   1:L PR[91] R[100]mm/sec CNT100;
   1:  PR[91,1] = PR[90,1] + 14.999;
   1:  PR[91,2] = PR[90,2] + -17.713;
   1:  PR[91,3] = PR[90,3] + 29.369;
   1:L PR[91] R[100]mm/sec CNT100;
   1:  PR[91,1] = PR[90,1] + 15.996;
   1:  PR[91,2] = PR[90,2] + -17.584;
   1:  PR[91,3] = PR[90,3] + 29.377;
   1:L PR[91] R[100]mm/sec CNT100;
   1:  PR[91,1] = PR[90,1] + 16.467;
   1:  PR[91,2] = PR[90,2] + -17.502;
   1:  PR[91,3] = PR[90,3] + 29.385;
   1:L PR[91] R[100]mm/sec CNT100;
   1:  PR[91,1] = PR[90,1] + 16.980;
   1:  PR[91,2] = PR[90,2] + -17.408;
   1:  PR[91,3] = PR[90,3] + 29.388;
   1:L PR[91] R[100]mm/sec CNT100;
   1:  PR[91,1] = PR[90,1] + 17.954;
   1:  PR[91,2] = PR[90,2] + -17.183;
   1:  PR[91,3] = PR[90,3] + 29.392;
   1:L PR[91] R[100]mm/sec CNT100;
   1:  PR[91,1] = PR[90,1] + 18.912;
   1:  PR[91,2] = PR[90,2] + -16.912;
   1:  PR[91,3] = PR[90,3] + 29.400;
   1:L PR[91] R[100]mm/sec CNT100;
   1:  PR[91,1] = PR[90,1] + 19.853;
   1:  PR[91,2] = PR[90,2] + -16.596;
   1:  PR[91,3] = PR[90,3] + 29.408;
   1:L PR[91] R[100]mm/sec CNT100;
   1:  PR[91,1] = PR[90,1] + 20.773;
   1:  PR[91,2] = PR[90,2] + -16.236;
   1:  PR[91,3] = PR[90,3] + 29.415;
   1:L PR[91] R[100]mm/sec CNT100;
   1:  PR[91,1] = PR[90,1] + 21.671;
   1:  PR[91,2] = PR[90,2] + -15.834;
   1:  PR[91,3] = PR[90,3] + 29.423;
   1:L PR[91] R[100]mm/sec CNT100;
   1:  PR[91,1] = PR[90,1] + 22.552;
   1:  PR[91,2] = PR[90,2] + -15.387;
   1:  PR[91,3] = PR[90,3] + 29.430;
   1:L PR[91] R[100]mm/sec CNT100;
   1:  PR[91,1] = PR[90,1] + 23.431;
   1:  PR[91,2] = PR[90,2] + -14.885;
   1:  PR[91,3] = PR[90,3] + 29.438;
   1:L PR[91] R[100]mm/sec CNT100;
   1:  PR[91,1] = PR[90,1] + 24.148;
   1:  PR[91,2] = PR[90,2] + -14.431;
   1:  PR[91,3] = PR[90,3] + 29.446;
   1:L PR[91] R[100]mm/sec CNT100;
   1:  PR[91,1] = PR[90,1] + 24.918;
   1:  PR[91,2] = PR[90,2] + -13.893;
   1:  PR[91,3] = PR[90,3] + 29.452;
   1:L PR[91] R[100]mm/sec CNT100;
   1:  PR[91,1] = PR[90,1] + 25.658;
   1:  PR[91,2] = PR[90,2] + -13.318;
   1:  PR[91,3] = PR[90,3] + 29.459;
   1:L PR[91] R[100]mm/sec CNT100;
   1:  PR[91,1] = PR[90,1] + 26.370;
   1:  PR[91,2] = PR[90,2] + -12.708;
   1:  PR[91,3] = PR[90,3] + 29.466;
   1:L PR[91] R[100]mm/sec CNT100;
   1:  PR[91,1] = PR[90,1] + 27.049;
   1:  PR[91,2] = PR[90,2] + -12.063;
   1:  PR[91,3] = PR[90,3] + 29.474;
   1:L PR[91] R[100]mm/sec CNT100;
   1:  PR[91,1] = PR[90,1] + 27.695;
   1:  PR[91,2] = PR[90,2] + -11.384;
   1:  PR[91,3] = PR[90,3] + 29.481;
   1:L PR[91] R[100]mm/sec CNT100;
   1:  PR[91,1] = PR[90,1] + 28.305;
   1:  PR[91,2] = PR[90,2] + -10.672;
   1:  PR[91,3] = PR[90,3] + 29.488;
   1:L PR[91] R[100]mm/sec CNT100;
   1:  PR[91,1] = PR[90,1] + 28.879;
   1:  PR[91,2] = PR[90,2] + -9.929;
   1:  PR[91,3] = PR[90,3] + 29.495;
   1:L PR[91] R[100]mm/sec CNT100;
   1:  PR[91,1] = PR[90,1] + 29.413;
   1:  PR[91,2] = PR[90,2] + -9.158;
   1:  PR[91,3] = PR[90,3] + 29.502;
   1:L PR[91] R[100]mm/sec CNT100;
   1:  PR[91,1] = PR[90,1] + 29.908;
   1:  PR[91,2] = PR[90,2] + -8.363;
   1:  PR[91,3] = PR[90,3] + 29.509;
   1:L PR[91] R[100]mm/sec CNT100;
   1:  PR[91,1] = PR[90,1] + 30.361;
   1:  PR[91,2] = PR[90,2] + -7.547;
   1:  PR[91,3] = PR[90,3] + 29.517;
   1:L PR[91] R[100]mm/sec CNT100;
   1:  PR[91,1] = PR[90,1] + 30.770;
   1:  PR[91,2] = PR[90,2] + -6.718;
   1:  PR[91,3] = PR[90,3] + 29.524;
   1:L PR[91] R[100]mm/sec CNT100;
   1:  PR[91,1] = PR[90,1] + 31.135;
   1:  PR[91,2] = PR[90,2] + -5.878;
   1:  PR[91,3] = PR[90,3] + 29.531;
   1:L PR[91] R[100]mm/sec CNT100;
   1:  PR[91,1] = PR[90,1] + 31.452;
   1:  PR[91,2] = PR[90,2] + -5.031;
   1:  PR[91,3] = PR[90,3] + 29.538;
   1:L PR[91] R[100]mm/sec CNT100;
   1:  PR[91,1] = PR[90,1] + 31.722;
   1:  PR[91,2] = PR[90,2] + -4.174;
   1:  PR[91,3] = PR[90,3] + 29.545;
   1:L PR[91] R[100]mm/sec CNT100;
   1:  PR[91,1] = PR[90,1] + 31.943;
   1:  PR[91,2] = PR[90,2] + -3.305;
   1:  PR[91,3] = PR[90,3] + 29.552;
   1:L PR[91] R[100]mm/sec CNT100;
   1:  PR[91,1] = PR[90,1] + 32.116;
   1:  PR[91,2] = PR[90,2] + -2.416;
   1:  PR[91,3] = PR[90,3] + 29.559;
   1:L PR[91] R[100]mm/sec CNT100;
   1:  PR[91,1] = PR[90,1] + 32.241;
   1:  PR[91,2] = PR[90,2] + -1.502;
   1:  PR[91,3] = PR[90,3] + 29.566;
   1:L PR[91] R[100]mm/sec CNT100;
   1:  PR[91,1] = PR[90,1] + 32.316;
   1:  PR[91,2] = PR[90,2] + -0.556;
   1:  PR[91,3] = PR[90,3] + 29.573;
   1:L PR[91] R[100]mm/sec CNT100;
   1:  PR[91,1] = PR[90,1] + 32.341;
   1:  PR[91,2] = PR[90,2] + 0.428;
   1:  PR[91,3] = PR[90,3] + 29.580;
   1:L PR[91] R[100]mm/sec CNT100;
   1:  PR[91,1] = PR[90,1] + 32.316;
   1:  PR[91,2] = PR[90,2] + 1.411;
   1:  PR[91,3] = PR[90,3] + 29.587;
   1:L PR[91] R[100]mm/sec CNT100;
   1:  PR[91,1] = PR[90,1] + 32.241;
   1:  PR[91,2] = PR[90,2] + 2.357;
   1:  PR[91,3] = PR[90,3] + 29.595;
   1:L PR[91] R[100]mm/sec CNT100;
   1:  PR[91,1] = PR[90,1] + 32.116;
   1:  PR[91,2] = PR[90,2] + 3.272;
   1:  PR[91,3] = PR[90,3] + 29.602;
   1:L PR[91] R[100]mm/sec CNT100;
   1:  PR[91,1] = PR[90,1] + 31.943;
   1:  PR[91,2] = PR[90,2] + 4.160;
   1:  PR[91,3] = PR[90,3] + 29.609;
   1:L PR[91] R[100]mm/sec CNT100;
   1:  PR[91,1] = PR[90,1] + 31.721;
   1:  PR[91,2] = PR[90,2] + 5.030;
   1:  PR[91,3] = PR[90,3] + 29.616;
   1:L PR[91] R[100]mm/sec CNT100;
   1:  PR[91,1] = PR[90,1] + 31.452;
   1:  PR[91,2] = PR[90,2] + 5.886;
   1:  PR[91,3] = PR[90,3] + 29.623;
   1:L PR[91] R[100]mm/sec CNT100;
   1:  PR[91,1] = PR[90,1] + 31.135;
   1:  PR[91,2] = PR[90,2] + 6.731;
   1:  PR[91,3] = PR[90,3] + 29.630;
   1:L PR[91] R[100]mm/sec CNT100;
   1:  PR[91,1] = PR[90,1] + 30.663;
   1:  PR[91,2] = PR[90,2] + 7.794;
   1:  PR[91,3] = PR[90,3] + 29.637;
   1:L PR[91] R[100]mm/sec CNT100;
   1:  PR[91,1] = PR[90,1] + 30.361;
   1:  PR[91,2] = PR[90,2] + 8.402;
   1:  PR[91,3] = PR[90,3] + 29.646;
   1:L PR[91] R[100]mm/sec CNT100;
   1:  PR[91,1] = PR[90,1] + 29.908;
   1:  PR[91,2] = PR[90,2] + 9.218;
   1:  PR[91,3] = PR[90,3] + 29.651;
   1:L PR[91] R[100]mm/sec CNT100;
   1:  PR[91,1] = PR[90,1] + 29.413;
   1:  PR[91,2] = PR[90,2] + 10.013;
   1:  PR[91,3] = PR[90,3] + 29.658;
   1:L PR[91] R[100]mm/sec CNT100;
   1:  PR[91,1] = PR[90,1] + 28.877;
   1:  PR[91,2] = PR[90,2] + 10.786;
   1:  PR[91,3] = PR[90,3] + 29.665;
   1:L PR[91] R[100]mm/sec CNT100;
   1:  PR[91,1] = PR[90,1] + 28.625;
   1:  PR[91,2] = PR[90,2] + 11.119;
   1:  PR[91,3] = PR[90,3] + 29.672;
   1:L PR[91] R[100]mm/sec CNT100;
   1:  PR[91,1] = PR[90,1] + 28.306;
   1:  PR[91,2] = PR[90,2] + 11.526;
   1:  PR[91,3] = PR[90,3] + 29.676;
   1:L PR[91] R[100]mm/sec CNT100;
   1:  PR[91,1] = PR[90,1] + 27.695;
   1:  PR[91,2] = PR[90,2] + 12.239;
   1:  PR[91,3] = PR[90,3] + 29.680;
   1:L PR[91] R[100]mm/sec CNT100;
   1:  PR[91,1] = PR[90,1] + 27.048;
   1:  PR[91,2] = PR[90,2] + 12.920;
   1:  PR[91,3] = PR[90,3] + 29.687;
   1:L PR[91] R[100]mm/sec CNT100;
   1:  PR[91,1] = PR[90,1] + 26.623;
   1:  PR[91,2] = PR[90,2] + 13.328;
   1:  PR[91,3] = PR[90,3] + 29.694;
   1:L PR[91] R[100]mm/sec CNT100;
   1:  PR[91,1] = PR[90,1] + 26.372;
   1:  PR[91,2] = PR[90,2] + 13.561;
   1:  PR[91,3] = PR[90,3] + 29.699;
   1:L PR[91] R[100]mm/sec CNT100;
   1:  PR[91,1] = PR[90,1] + 25.658;
   1:  PR[91,2] = PR[90,2] + 14.173;
   1:  PR[91,3] = PR[90,3] + 29.701;
   1:L PR[91] R[100]mm/sec CNT100;
   1:  PR[91,1] = PR[90,1] + 24.917;
   1:  PR[91,2] = PR[90,2] + 14.748;
   1:  PR[91,3] = PR[90,3] + 29.708;
   1:L PR[91] R[100]mm/sec CNT100;
   1:  PR[91,1] = PR[90,1] + 24.280;
   1:  PR[91,2] = PR[90,2] + 15.197;
   1:  PR[91,3] = PR[90,3] + 29.716;
   1:L PR[91] R[100]mm/sec CNT100;
   1:  PR[91,1] = PR[90,1] + 23.430;
   1:  PR[91,2] = PR[90,2] + 15.741;
   1:  PR[91,3] = PR[90,3] + 29.721;
   1:L PR[91] R[100]mm/sec CNT100;
   1:  PR[91,1] = PR[90,1] + 22.536;
   1:  PR[91,2] = PR[90,2] + 16.250;
   1:  PR[91,3] = PR[90,3] + 29.729;
   1:L PR[91] R[100]mm/sec CNT100;
   1:  PR[91,1] = PR[90,1] + 21.672;
   1:  PR[91,2] = PR[90,2] + 16.689;
   1:  PR[91,3] = PR[90,3] + 29.737;
   1:L PR[91] R[100]mm/sec CNT100;
   1:  PR[91,1] = PR[90,1] + 20.773;
   1:  PR[91,2] = PR[90,2] + 17.091;
   1:  PR[91,3] = PR[90,3] + 29.745;
   1:L PR[91] R[100]mm/sec CNT100;
   1:  PR[91,1] = PR[90,1] + 20.033;
   1:  PR[91,2] = PR[90,2] + 17.382;
   1:  PR[91,3] = PR[90,3] + 29.752;
   1:L PR[91] R[100]mm/sec CNT100;
   1:  PR[91,1] = PR[90,1] + 18.911;
   1:  PR[91,2] = PR[90,2] + 17.768;
   1:  PR[91,3] = PR[90,3] + 29.758;
   1:L PR[91] R[100]mm/sec CNT100;
   1:  PR[91,1] = PR[90,1] + 17.954;
   1:  PR[91,2] = PR[90,2] + 18.038;
   1:  PR[91,3] = PR[90,3] + 29.767;
   1:L PR[91] R[100]mm/sec CNT100;
   1:  PR[91,1] = PR[90,1] + 16.981;
   1:  PR[91,2] = PR[90,2] + 18.263;
   1:  PR[91,3] = PR[90,3] + 29.775;
   1:L PR[91] R[100]mm/sec CNT100;
   1:  PR[91,1] = PR[90,1] + 15.995;
   1:  PR[91,2] = PR[90,2] + 18.440;
   1:  PR[91,3] = PR[90,3] + 29.783;
   1:L PR[91] R[100]mm/sec CNT100;
   1:  PR[91,1] = PR[90,1] + 14.997;
   1:  PR[91,2] = PR[90,2] + 18.568;
   1:  PR[91,3] = PR[90,3] + 29.790;
   1:L PR[91] R[100]mm/sec CNT100;
   1:  PR[91,1] = PR[90,1] + 14.620;
   1:  PR[91,2] = PR[90,2] + 18.600;
   1:  PR[91,3] = PR[90,3] + 29.798;
   1:L PR[91] R[100]mm/sec CNT100;
   1:  PR[91,1] = PR[90,1] + 13.996;
   1:  PR[91,2] = PR[90,2] + 18.647;
   1:  PR[91,3] = PR[90,3] + 29.801;
   1:L PR[91] R[100]mm/sec CNT100;
   1:  PR[91,1] = PR[90,1] + 12.987;
   1:  PR[91,2] = PR[90,2] + 18.676;
   1:  PR[91,3] = PR[90,3] + 29.806;
   1:L PR[91] R[100]mm/sec CNT100;
   1:  PR[91,1] = PR[90,1] + 11.977;
   1:  PR[91,2] = PR[90,2] + 18.656;
   1:  PR[91,3] = PR[90,3] + 29.813;
   1:L PR[91] R[100]mm/sec CNT100;
   1:  PR[91,1] = PR[90,1] + 10.968;
   1:  PR[91,2] = PR[90,2] + 18.586;
   1:  PR[91,3] = PR[90,3] + 29.821;
   1:L PR[91] R[100]mm/sec CNT100;
   1:  PR[91,1] = PR[90,1] + 9.963;
   1:  PR[91,2] = PR[90,2] + 18.465;
   1:  PR[91,3] = PR[90,3] + 29.829;
   1:L PR[91] R[100]mm/sec CNT100;
   1:  PR[91,1] = PR[90,1] + 8.960;
   1:  PR[91,2] = PR[90,2] + 18.294;
   1:  PR[91,3] = PR[90,3] + 29.837;
   1:L PR[91] R[100]mm/sec CNT100;
   1:  PR[91,1] = PR[90,1] + 7.961;
   1:  PR[91,2] = PR[90,2] + 18.072;
   1:  PR[91,3] = PR[90,3] + 29.844;
   1:L PR[91] R[100]mm/sec CNT100;
   1:  PR[91,1] = PR[90,1] + 6.974;
   1:  PR[91,2] = PR[90,2] + 17.799;
   1:  PR[91,3] = PR[90,3] + 29.852;
   1:L PR[91] R[100]mm/sec CNT100;
   1:  PR[91,1] = PR[90,1] + 6.001;
   1:  PR[91,2] = PR[90,2] + 17.476;
   1:  PR[91,3] = PR[90,3] + 29.860;
   1:L PR[91] R[100]mm/sec CNT100;
   1:  PR[91,1] = PR[90,1] + 5.327;
   1:  PR[91,2] = PR[90,2] + 17.218;
   1:  PR[91,3] = PR[90,3] + 29.868;
   1:L PR[91] R[100]mm/sec CNT100;
   1:  PR[91,1] = PR[90,1] + 4.116;
   1:  PR[91,2] = PR[90,2] + 16.684;
   1:  PR[91,3] = PR[90,3] + 29.873;
   1:L PR[91] R[100]mm/sec CNT100;
   1:  PR[91,1] = PR[90,1] + 3.212;
   1:  PR[91,2] = PR[90,2] + 16.219;
   1:  PR[91,3] = PR[90,3] + 29.884;
   1:L PR[91] R[100]mm/sec CNT100;
   1:  PR[91,1] = PR[90,1] + 2.333;
   1:  PR[91,2] = PR[90,2] + 15.706;
   1:  PR[91,3] = PR[90,3] + 29.891;
   1:L PR[91] R[100]mm/sec CNT100;
   1:  PR[91,1] = PR[90,1] + 1.446;
   1:  PR[91,2] = PR[90,2] + 15.121;
   1:  PR[91,3] = PR[90,3] + 29.899;
   1:L PR[91] R[100]mm/sec CNT100;
   1:  PR[91,1] = PR[90,1] + 1.018;
   1:  PR[91,2] = PR[90,2] + 14.899;
   1:  PR[91,3] = PR[90,3] + 29.907;
   1:L PR[91] R[100]mm/sec CNT100;
   1:  PR[91,1] = PR[90,1] + 0.546;
   1:  PR[91,2] = PR[90,2] + 14.747;
   1:  PR[91,3] = PR[90,3] + 29.911;
   1:L PR[91] R[100]mm/sec CNT100;
   1:  PR[91,1] = PR[90,1] + 0.057;
   1:  PR[91,2] = PR[90,2] + 14.675;
   1:  PR[91,3] = PR[90,3] + 29.915;
   1:L PR[91] R[100]mm/sec CNT100;
   1:  PR[91,1] = PR[90,1] + -0.437;
   1:  PR[91,2] = PR[90,2] + 14.686;
   1:  PR[91,3] = PR[90,3] + 29.919;
   1:L PR[91] R[100]mm/sec CNT100;
   1:  PR[91,1] = PR[90,1] + -0.921;
   1:  PR[91,2] = PR[90,2] + 14.781;
   1:  PR[91,3] = PR[90,3] + 29.922;
   1:L PR[91] R[100]mm/sec CNT100;
   1:  PR[91,1] = PR[90,1] + -1.380;
   1:  PR[91,2] = PR[90,2] + 14.954;
   1:  PR[91,3] = PR[90,3] + 29.926;
   1:L PR[91] R[100]mm/sec CNT100;
   1:  PR[91,1] = PR[90,1] + -1.780;
   1:  PR[91,2] = PR[90,2] + 15.184;
   1:  PR[91,3] = PR[90,3] + 29.930;
   1:L PR[91] R[100]mm/sec CNT100;
   1:  PR[91,1] = PR[90,1] + -2.575;
   1:  PR[91,2] = PR[90,2] + 15.706;
   1:  PR[91,3] = PR[90,3] + 29.933;
   1:L PR[91] R[100]mm/sec CNT100;
   1:  PR[91,1] = PR[90,1] + -3.455;
   1:  PR[91,2] = PR[90,2] + 16.219;
   1:  PR[91,3] = PR[90,3] + 29.941;
   1:L PR[91] R[100]mm/sec CNT100;
   1:  PR[91,1] = PR[90,1] + -4.361;
   1:  PR[91,2] = PR[90,2] + 16.686;
   1:  PR[91,3] = PR[90,3] + 29.948;
   1:L PR[91] R[100]mm/sec CNT100;
   1:  PR[91,1] = PR[90,1] + -5.291;
   1:  PR[91,2] = PR[90,2] + 17.106;
   1:  PR[91,3] = PR[90,3] + 29.956;
   1:L PR[91] R[100]mm/sec CNT100;
   1:  PR[91,1] = PR[90,1] + -6.465;
   1:  PR[91,2] = PR[90,2] + 17.557;
   1:  PR[91,3] = PR[90,3] + 29.964;
   1:L PR[91] R[100]mm/sec CNT100;
   1:  PR[91,1] = PR[90,1] + -7.374;
   1:  PR[91,2] = PR[90,2] + 17.849;
   1:  PR[91,3] = PR[90,3] + 29.974;
   1:L PR[91] R[100]mm/sec CNT100;
   1:  PR[91,1] = PR[90,1] + -8.297;
   1:  PR[91,2] = PR[90,2] + 18.097;
   1:  PR[91,3] = PR[90,3] + 29.981;
   1:L PR[91] R[100]mm/sec CNT100;
   1:  PR[91,1] = PR[90,1] + -9.229;
   1:  PR[91,2] = PR[90,2] + 18.301;
   1:  PR[91,3] = PR[90,3] + 29.988;
   1:L PR[91] R[100]mm/sec CNT100;
   1:  PR[91,1] = PR[90,1] + -10.173;
   1:  PR[91,2] = PR[90,2] + 18.461;
   1:  PR[91,3] = PR[90,3] + 29.996;
   1:L PR[91] R[100]mm/sec CNT100;
   1:  PR[91,1] = PR[90,1] + -11.242;
   1:  PR[91,2] = PR[90,2] + 18.589;
   1:  PR[91,3] = PR[90,3] + 30.003;
   1:L PR[91] R[100]mm/sec CNT100;
   1:  PR[91,1] = PR[90,1] + -12.277;
   1:  PR[91,2] = PR[90,2] + 18.658;
   1:  PR[91,3] = PR[90,3] + 30.011;
   1:L PR[91] R[100]mm/sec CNT100;
   1:  PR[91,1] = PR[90,1] + -13.317;
   1:  PR[91,2] = PR[90,2] + 18.674;
   1:  PR[91,3] = PR[90,3] + 30.019;
   1:L PR[91] R[100]mm/sec CNT100;
   1:  PR[91,1] = PR[90,1] + -14.358;
   1:  PR[91,2] = PR[90,2] + 18.638;
   1:  PR[91,3] = PR[90,3] + 30.027;
   1:L PR[91] R[100]mm/sec CNT100;
   1:  PR[91,1] = PR[90,1] + -15.398;
   1:  PR[91,2] = PR[90,2] + 18.548;
   1:  PR[91,3] = PR[90,3] + 30.035;
   1:L PR[91] R[100]mm/sec CNT100;
   1:  PR[91,1] = PR[90,1] + -16.433;
   1:  PR[91,2] = PR[90,2] + 18.406;
   1:  PR[91,3] = PR[90,3] + 30.043;
   1:L PR[91] R[100]mm/sec CNT100;
   1:  PR[91,1] = PR[90,1] + -17.461;
   1:  PR[91,2] = PR[90,2] + 18.210;
   1:  PR[91,3] = PR[90,3] + 30.051;
   1:L PR[91] R[100]mm/sec CNT100;
   1:  PR[91,1] = PR[90,1] + -18.477;
   1:  PR[91,2] = PR[90,2] + 17.963;
   1:  PR[91,3] = PR[90,3] + 30.059;
   1:L PR[91] R[100]mm/sec CNT100;
   1:  PR[91,1] = PR[90,1] + -19.479;
   1:  PR[91,2] = PR[90,2] + 17.663;
   1:  PR[91,3] = PR[90,3] + 30.067;
   1:L PR[91] R[100]mm/sec CNT100;
   1:  PR[91,1] = PR[90,1] + -20.464;
   1:  PR[91,2] = PR[90,2] + 17.312;
   1:  PR[91,3] = PR[90,3] + 30.075;
   1:L PR[91] R[100]mm/sec CNT100;
   1:  PR[91,1] = PR[90,1] + -21.512;
   1:  PR[91,2] = PR[90,2] + 16.874;
   1:  PR[91,3] = PR[90,3] + 30.083;
   1:L PR[91] R[100]mm/sec CNT100;
   1:  PR[91,1] = PR[90,1] + -22.383;
   1:  PR[91,2] = PR[90,2] + 16.454;
   1:  PR[91,3] = PR[90,3] + 30.092;
   1:L PR[91] R[100]mm/sec CNT100;
   1:  PR[91,1] = PR[90,1] + -23.252;
   1:  PR[91,2] = PR[90,2] + 15.985;
   1:  PR[91,3] = PR[90,3] + 30.099;
   1:L PR[91] R[100]mm/sec CNT100;
   1:  PR[91,1] = PR[90,1] + -24.098;
   1:  PR[91,2] = PR[90,2] + 15.473;
   1:  PR[91,3] = PR[90,3] + 30.107;
   1:L PR[91] R[100]mm/sec CNT100;
   1:  PR[91,1] = PR[90,1] + -24.912;
   1:  PR[91,2] = PR[90,2] + 14.922;
   1:  PR[91,3] = PR[90,3] + 30.114;
   1:L PR[91] R[100]mm/sec CNT100;
   1:  PR[91,1] = PR[90,1] + -25.694;
   1:  PR[91,2] = PR[90,2] + 14.334;
   1:  PR[91,3] = PR[90,3] + 30.122;
   1:L PR[91] R[100]mm/sec CNT100;
   1:  PR[91,1] = PR[90,1] + -26.442;
   1:  PR[91,2] = PR[90,2] + 13.710;
   1:  PR[91,3] = PR[90,3] + 30.129;
   1:L PR[91] R[100]mm/sec CNT100;
   1:  PR[91,1] = PR[90,1] + -27.153;
   1:  PR[91,2] = PR[90,2] + 13.052;
   1:  PR[91,3] = PR[90,3] + 30.137;
   1:L PR[91] R[100]mm/sec CNT100;
   1:  PR[91,1] = PR[90,1] + -27.826;
   1:  PR[91,2] = PR[90,2] + 12.360;
   1:  PR[91,3] = PR[90,3] + 30.144;
   1:L PR[91] R[100]mm/sec CNT100;
   1:  PR[91,1] = PR[90,1] + -28.460;
   1:  PR[91,2] = PR[90,2] + 11.637;
   1:  PR[91,3] = PR[90,3] + 30.152;
   1:L PR[91] R[100]mm/sec CNT100;
   1:  PR[91,1] = PR[90,1] + -29.053;
   1:  PR[91,2] = PR[90,2] + 10.882;
   1:  PR[91,3] = PR[90,3] + 30.159;
   1:L PR[91] R[100]mm/sec CNT100;
   1:  PR[91,1] = PR[90,1] + -29.603;
   1:  PR[91,2] = PR[90,2] + 10.098;
   1:  PR[91,3] = PR[90,3] + 30.166;
   1:L PR[91] R[100]mm/sec CNT100;
   1:  PR[91,1] = PR[90,1] + -30.110;
   1:  PR[91,2] = PR[90,2] + 9.289;
   1:  PR[91,3] = PR[90,3] + 30.174;
   1:L PR[91] R[100]mm/sec CNT100;
   1:  PR[91,1] = PR[90,1] + -30.573;
   1:  PR[91,2] = PR[90,2] + 8.458;
   1:  PR[91,3] = PR[90,3] + 30.181;
   1:L PR[91] R[100]mm/sec CNT100;
   1:  PR[91,1] = PR[90,1] + -30.990;
   1:  PR[91,2] = PR[90,2] + 7.611;
   1:  PR[91,3] = PR[90,3] + 30.188;
   1:L PR[91] R[100]mm/sec CNT100;
   1:  PR[91,1] = PR[90,1] + -31.360;
   1:  PR[91,2] = PR[90,2] + 6.755;
   1:  PR[91,3] = PR[90,3] + 30.196;
   1:L PR[91] R[100]mm/sec CNT100;
   1:  PR[91,1] = PR[90,1] + -31.682;
   1:  PR[91,2] = PR[90,2] + 5.894;
   1:  PR[91,3] = PR[90,3] + 30.203;
   1:L PR[91] R[100]mm/sec CNT100;
   1:  PR[91,1] = PR[90,1] + -31.955;
   1:  PR[91,2] = PR[90,2] + 5.028;
   1:  PR[91,3] = PR[90,3] + 30.210;
   1:L PR[91] R[100]mm/sec CNT100;
   1:  PR[91,1] = PR[90,1] + -32.179;
   1:  PR[91,2] = PR[90,2] + 4.154;
   1:  PR[91,3] = PR[90,3] + 30.217;
   1:L PR[91] R[100]mm/sec CNT100;
   1:  PR[91,1] = PR[90,1] + -32.354;
   1:  PR[91,2] = PR[90,2] + 3.267;
   1:  PR[91,3] = PR[90,3] + 30.224;
   1:L PR[91] R[100]mm/sec CNT100;
   1:  PR[91,1] = PR[90,1] + -32.479;
   1:  PR[91,2] = PR[90,2] + 2.356;
   1:  PR[91,3] = PR[90,3] + 30.231;
   1:L PR[91] R[100]mm/sec CNT100;
   1:  PR[91,1] = PR[90,1] + -32.555;
   1:  PR[91,2] = PR[90,2] + 1.412;
   1:  PR[91,3] = PR[90,3] + 30.238;
   1:L PR[91] R[100]mm/sec CNT100;
   1:  PR[91,1] = PR[90,1] + -32.580;
   1:  PR[91,2] = PR[90,2] + 0.428;
   1:  PR[91,3] = PR[90,3] + 30.245;
   1:L PR[91] R[100]mm/sec CNT100;
   1:  PR[91,1] = PR[90,1] + -32.555;
   1:  PR[91,2] = PR[90,2] + -0.557;
   1:  PR[91,3] = PR[90,3] + 30.252;
   1:L PR[91] R[100]mm/sec CNT100;
   1:  PR[91,1] = PR[90,1] + -32.479;
   1:  PR[91,2] = PR[90,2] + -1.500;
   1:  PR[91,3] = PR[90,3] + 30.260;
   1:L PR[91] R[100]mm/sec CNT100;
   1:  PR[91,1] = PR[90,1] + -32.354;
   1:  PR[91,2] = PR[90,2] + -2.412;
   1:  PR[91,3] = PR[90,3] + 30.267;
   1:L PR[91] R[100]mm/sec CNT100;
   1:  PR[91,1] = PR[90,1] + -32.179;
   1:  PR[91,2] = PR[90,2] + -3.299;
   1:  PR[91,3] = PR[90,3] + 30.274;
   1:L PR[91] R[100]mm/sec CNT100;
   1:  PR[91,1] = PR[90,1] + -31.956;
   1:  PR[91,2] = PR[90,2] + -4.172;
   1:  PR[91,3] = PR[90,3] + 30.281;
   1:L PR[91] R[100]mm/sec CNT100;
   1:  PR[91,1] = PR[90,1] + -31.682;
   1:  PR[91,2] = PR[90,2] + -5.039;
   1:  PR[91,3] = PR[90,3] + 30.288;
   1:L PR[91] R[100]mm/sec CNT100;
   1:  PR[91,1] = PR[90,1] + -31.360;
   1:  PR[91,2] = PR[90,2] + -5.900;
   1:  PR[91,3] = PR[90,3] + 30.295;
   1:L PR[91] R[100]mm/sec CNT100;
   1:  PR[91,1] = PR[90,1] + -30.990;
   1:  PR[91,2] = PR[90,2] + -6.756;
   1:  PR[91,3] = PR[90,3] + 30.302;
   1:L PR[91] R[100]mm/sec CNT100;
   1:  PR[91,1] = PR[90,1] + -30.573;
   1:  PR[91,2] = PR[90,2] + -7.603;
   1:  PR[91,3] = PR[90,3] + 30.309;
   1:L PR[91] R[100]mm/sec CNT100;
   1:  PR[91,1] = PR[90,1] + -30.110;
   1:  PR[91,2] = PR[90,2] + -8.434;
   1:  PR[91,3] = PR[90,3] + 30.316;
   1:L PR[91] R[100]mm/sec CNT100;
   1:  PR[91,1] = PR[90,1] + -29.603;
   1:  PR[91,2] = PR[90,2] + -9.243;
   1:  PR[91,3] = PR[90,3] + 30.324;
   1:L PR[91] R[100]mm/sec CNT100;
   1:  PR[91,1] = PR[90,1] + -29.053;
   1:  PR[91,2] = PR[90,2] + -10.027;
   1:  PR[91,3] = PR[90,3] + 30.331;
   1:L PR[91] R[100]mm/sec CNT100;
   1:  PR[91,1] = PR[90,1] + -28.460;
   1:  PR[91,2] = PR[90,2] + -10.781;
   1:  PR[91,3] = PR[90,3] + 30.338;
   1:L PR[91] R[100]mm/sec CNT100;
   1:  PR[91,1] = PR[90,1] + -27.826;
   1:  PR[91,2] = PR[90,2] + -11.505;
   1:  PR[91,3] = PR[90,3] + 30.346;
   1:L PR[91] R[100]mm/sec CNT100;
   1:  PR[91,1] = PR[90,1] + -27.153;
   1:  PR[91,2] = PR[90,2] + -12.197;
   1:  PR[91,3] = PR[90,3] + 30.353;
   1:L PR[91] R[100]mm/sec CNT100;
   1:  PR[91,1] = PR[90,1] + -26.442;
   1:  PR[91,2] = PR[90,2] + -12.855;
   1:  PR[91,3] = PR[90,3] + 30.360;
   1:L PR[91] R[100]mm/sec CNT100;
   1:  PR[91,1] = PR[90,1] + -25.694;
   1:  PR[91,2] = PR[90,2] + -13.479;
   1:  PR[91,3] = PR[90,3] + 30.368;
   1:L PR[91] R[100]mm/sec CNT100;
   1:  PR[91,1] = PR[90,1] + -24.912;
   1:  PR[91,2] = PR[90,2] + -14.067;
   1:  PR[91,3] = PR[90,3] + 30.375;
   1:L PR[91] R[100]mm/sec CNT100;
   1:  PR[91,1] = PR[90,1] + -24.098;
   1:  PR[91,2] = PR[90,2] + -14.617;
   1:  PR[91,3] = PR[90,3] + 30.383;
   1:L PR[91] R[100]mm/sec CNT100;
   1:  PR[91,1] = PR[90,1] + -23.252;
   1:  PR[91,2] = PR[90,2] + -15.129;
   1:  PR[91,3] = PR[90,3] + 30.390;
   1:L PR[91] R[100]mm/sec CNT100;
   1:  PR[91,1] = PR[90,1] + -22.370;
   1:  PR[91,2] = PR[90,2] + -15.606;
   1:  PR[91,3] = PR[90,3] + 30.398;
   1:L PR[91] R[100]mm/sec CNT100;
   1:  PR[91,1] = PR[90,1] + -21.427;
   1:  PR[91,2] = PR[90,2] + -16.057;
   1:  PR[91,3] = PR[90,3] + 30.406;
   1:L PR[91] R[100]mm/sec CNT100;
   1:  PR[91,1] = PR[90,1] + -20.622;
   1:  PR[91,2] = PR[90,2] + -16.396;
   1:  PR[91,3] = PR[90,3] + 30.414;
   1:L PR[91] R[100]mm/sec CNT100;
   1:  PR[91,1] = PR[90,1] + -19.478;
   1:  PR[91,2] = PR[90,2] + -16.808;
   1:  PR[91,3] = PR[90,3] + 30.420;
   1:L PR[91] R[100]mm/sec CNT100;
   1:  PR[91,1] = PR[90,1] + -18.477;
   1:  PR[91,2] = PR[90,2] + -17.107;
   1:  PR[91,3] = PR[90,3] + 30.430;
   1:L PR[91] R[100]mm/sec CNT100;
   1:  PR[91,1] = PR[90,1] + -17.461;
   1:  PR[91,2] = PR[90,2] + -17.355;
   1:  PR[91,3] = PR[90,3] + 30.438;
   1:L PR[91] R[100]mm/sec CNT100;
   1:  PR[91,1] = PR[90,1] + -16.433;
   1:  PR[91,2] = PR[90,2] + -17.550;
   1:  PR[91,3] = PR[90,3] + 30.446;
   1:L PR[91] R[100]mm/sec CNT100;
   1:  PR[91,1] = PR[90,1] + -15.398;
   1:  PR[91,2] = PR[90,2] + -17.693;
   1:  PR[91,3] = PR[90,3] + 30.454;
   1:L PR[91] R[100]mm/sec CNT100;
   1:  PR[91,1] = PR[90,1] + -14.358;
   1:  PR[91,2] = PR[90,2] + -17.783;
   1:  PR[91,3] = PR[90,3] + 30.462;
   1:L PR[91] R[100]mm/sec CNT100;
   1:  PR[91,1] = PR[90,1] + -13.317;
   1:  PR[91,2] = PR[90,2] + -17.819;
   1:  PR[91,3] = PR[90,3] + 30.470;
   1:L PR[91] R[100]mm/sec CNT100;
   1:  PR[91,1] = PR[90,1] + -12.278;
   1:  PR[91,2] = PR[90,2] + -17.803;
   1:  PR[91,3] = PR[90,3] + 30.478;
   1:L PR[91] R[100]mm/sec CNT100;
   1:  PR[91,1] = PR[90,1] + -11.244;
   1:  PR[91,2] = PR[90,2] + -17.734;
   1:  PR[91,3] = PR[90,3] + 30.486;
   1:L PR[91] R[100]mm/sec CNT100;
   1:  PR[91,1] = PR[90,1] + -10.174;
   1:  PR[91,2] = PR[90,2] + -17.606;
   1:  PR[91,3] = PR[90,3] + 30.493;
   1:L PR[91] R[100]mm/sec CNT100;
   1:  PR[91,1] = PR[90,1] + -9.202;
   1:  PR[91,2] = PR[90,2] + -17.441;
   1:  PR[91,3] = PR[90,3] + 30.502;
   1:L PR[91] R[100]mm/sec CNT100;
   1:  PR[91,1] = PR[90,1] + -8.202;
   1:  PR[91,2] = PR[90,2] + -17.219;
   1:  PR[91,3] = PR[90,3] + 30.509;
   1:L PR[91] R[100]mm/sec CNT100;
   1:  PR[91,1] = PR[90,1] + -7.376;
   1:  PR[91,2] = PR[90,2] + -16.994;
   1:  PR[91,3] = PR[90,3] + 30.517;
   1:L PR[91] R[100]mm/sec CNT100;
   1:  PR[91,1] = PR[90,1] + -6.464;
   1:  PR[91,2] = PR[90,2] + -16.701;
   1:  PR[91,3] = PR[90,3] + 30.524;
   1:L PR[91] R[100]mm/sec CNT100;
   1:  PR[91,1] = PR[90,1] + -5.568;
   1:  PR[91,2] = PR[90,2] + -16.365;
   1:  PR[91,3] = PR[90,3] + 30.531;
   1:L PR[91] R[100]mm/sec CNT100;
   1:  PR[91,1] = PR[90,1] + -4.360;
   1:  PR[91,2] = PR[90,2] + -15.831;
   1:  PR[91,3] = PR[90,3] + 30.538;
   1:L PR[91] R[100]mm/sec CNT100;
   1:  PR[91,1] = PR[90,1] + -3.455;
   1:  PR[91,2] = PR[90,2] + -15.364;
   1:  PR[91,3] = PR[90,3] + 30.548;
   1:L PR[91] R[100]mm/sec CNT100;
   1:  PR[91,1] = PR[90,1] + -2.576;
   1:  PR[91,2] = PR[90,2] + -14.851;
   1:  PR[91,3] = PR[90,3] + 30.556;
   1:L PR[91] R[100]mm/sec CNT100;
   1:  PR[91,1] = PR[90,1] + -1.780;
   1:  PR[91,2] = PR[90,2] + -14.329;
   1:  PR[91,3] = PR[90,3] + 30.564;
   1:L PR[91] R[100]mm/sec CNT100;
   1:  PR[91,1] = PR[90,1] + -1.381;
   1:  PR[91,2] = PR[90,2] + -14.099;
   1:  PR[91,3] = PR[90,3] + 30.571;
   1:L PR[91] R[100]mm/sec CNT100;
   1:  PR[91,1] = PR[90,1] + -0.921;
   1:  PR[91,2] = PR[90,2] + -13.926;
   1:  PR[91,3] = PR[90,3] + 30.575;
   1:L PR[91] R[100]mm/sec CNT100;
   1:  PR[91,1] = PR[90,1] + -0.437;
   1:  PR[91,2] = PR[90,2] + -13.831;
   1:  PR[91,3] = PR[90,3] + 30.579;
   1:L PR[91] R[100]mm/sec CNT100;
   1:  PR[91,1] = PR[90,1] + 0.057;
   1:  PR[91,2] = PR[90,2] + -13.820;
   1:  PR[91,3] = PR[90,3] + 30.582;
   1:L PR[91] R[100]mm/sec CNT100;
   1:  PR[91,1] = PR[90,1] + 0.546;
   1:  PR[91,2] = PR[90,2] + -13.891;
   1:  PR[91,3] = PR[90,3] + 30.586;
   1:L PR[91] R[100]mm/sec CNT100;
   1:  PR[91] = PR[90];
   1:  PR[91,1] = PR[90,1] + 1.102;
   1:  PR[91,2] = PR[90,2] + -14.607;
   1:  PR[91,3] = PR[90,3] + 31.920;
   1:L PR[91] R[100]mm/sec CNT100;
   1:  PR[91,1] = PR[90,1] + 1.462;
   1:  PR[91,2] = PR[90,2] + -14.803;
   1:  PR[91,3] = PR[90,3] + 30.594;
   1:L PR[91] R[100]mm/sec CNT100;
   1:  PR[91,1] = PR[90,1] + 2.356;
   1:  PR[91,2] = PR[90,2] + -15.345;
   1:  PR[91,3] = PR[90,3] + 30.597;
   1:L PR[91] R[100]mm/sec CNT100;
   1:  PR[91,1] = PR[90,1] + 3.212;
   1:  PR[91,2] = PR[90,2] + -15.805;
   1:  PR[91,3] = PR[90,3] + 30.605;
   1:L PR[91] R[100]mm/sec CNT100;
   1:  PR[91,1] = PR[90,1] + 4.293;
   1:  PR[91,2] = PR[90,2] + -16.311;
   1:  PR[91,3] = PR[90,3] + 30.613;
   1:L PR[91] R[100]mm/sec CNT100;
   1:  PR[91,1] = PR[90,1] + 5.250;
   1:  PR[91,2] = PR[90,2] + -16.696;
   1:  PR[91,3] = PR[90,3] + 30.622;
   1:L PR[91] R[100]mm/sec CNT100;
   1:  PR[91,1] = PR[90,1] + 6.230;
   1:  PR[91,2] = PR[90,2] + -17.033;
   1:  PR[91,3] = PR[90,3] + 30.630;
   1:L PR[91] R[100]mm/sec CNT100;
   1:  PR[91,1] = PR[90,1] + 6.835;
   1:  PR[91,2] = PR[90,2] + -17.212;
   1:  PR[91,3] = PR[90,3] + 30.638;
   1:L PR[91] R[100]mm/sec CNT100;
   1:  PR[91,1] = PR[90,1] + 7.218;
   1:  PR[91,2] = PR[90,2] + -17.317;
   1:  PR[91,3] = PR[90,3] + 30.643;
   1:L PR[91] R[100]mm/sec CNT100;
   1:  PR[91,1] = PR[90,1] + 8.229;
   1:  PR[91,2] = PR[90,2] + -17.552;
   1:  PR[91,3] = PR[90,3] + 30.646;
   1:L PR[91] R[100]mm/sec CNT100;
   1:  PR[91,1] = PR[90,1] + 9.246;
   1:  PR[91,2] = PR[90,2] + -17.734;
   1:  PR[91,3] = PR[90,3] + 30.654;
   1:L PR[91] R[100]mm/sec CNT100;
   1:  PR[91,1] = PR[90,1] + 10.271;
   1:  PR[91,2] = PR[90,2] + -17.864;
   1:  PR[91,3] = PR[90,3] + 30.662;
   1:L PR[91] R[100]mm/sec CNT100;
   1:  PR[91,1] = PR[90,1] + 11.299;
   1:  PR[91,2] = PR[90,2] + -17.942;
   1:  PR[91,3] = PR[90,3] + 30.670;
   1:L PR[91] R[100]mm/sec CNT100;
   1:  PR[91,1] = PR[90,1] + 12.329;
   1:  PR[91,2] = PR[90,2] + -17.968;
   1:  PR[91,3] = PR[90,3] + 30.678;
   1:L PR[91] R[100]mm/sec CNT100;
   1:  PR[91,1] = PR[90,1] + 13.356;
   1:  PR[91,2] = PR[90,2] + -17.942;
   1:  PR[91,3] = PR[90,3] + 30.686;
   1:L PR[91] R[100]mm/sec CNT100;
   1:  PR[91,1] = PR[90,1] + 14.378;
   1:  PR[91,2] = PR[90,2] + -17.865;
   1:  PR[91,3] = PR[90,3] + 30.694;
   1:L PR[91] R[100]mm/sec CNT100;
   1:  PR[91,1] = PR[90,1] + 15.393;
   1:  PR[91,2] = PR[90,2] + -17.737;
   1:  PR[91,3] = PR[90,3] + 30.702;
   1:L PR[91] R[100]mm/sec CNT100;
   1:  PR[91,1] = PR[90,1] + 16.390;
   1:  PR[91,2] = PR[90,2] + -17.563;
   1:  PR[91,3] = PR[90,3] + 30.710;
   1:L PR[91] R[100]mm/sec CNT100;
   1:  PR[91,1] = PR[90,1] + 17.372;
   1:  PR[91,2] = PR[90,2] + -17.341;
   1:  PR[91,3] = PR[90,3] + 30.717;
   1:L PR[91] R[100]mm/sec CNT100;
   1:  PR[91,1] = PR[90,1] + 18.340;
   1:  PR[91,2] = PR[90,2] + -17.072;
   1:  PR[91,3] = PR[90,3] + 30.725;
   1:L PR[91] R[100]mm/sec CNT100;
   1:  PR[91,1] = PR[90,1] + 19.291;
   1:  PR[91,2] = PR[90,2] + -16.756;
   1:  PR[91,3] = PR[90,3] + 30.733;
   1:L PR[91] R[100]mm/sec CNT100;
   1:  PR[91,1] = PR[90,1] + 20.221;
   1:  PR[91,2] = PR[90,2] + -16.396;
   1:  PR[91,3] = PR[90,3] + 30.741;
   1:L PR[91] R[100]mm/sec CNT100;
   1:  PR[91,1] = PR[90,1] + 21.128;
   1:  PR[91,2] = PR[90,2] + -15.993;
   1:  PR[91,3] = PR[90,3] + 30.748;
   1:L PR[91] R[100]mm/sec CNT100;
   1:  PR[91,1] = PR[90,1] + 22.012;
   1:  PR[91,2] = PR[90,2] + -15.548;
   1:  PR[91,3] = PR[90,3] + 30.756;
   1:L PR[91] R[100]mm/sec CNT100;
   1:  PR[91,1] = PR[90,1] + 22.868;
   1:  PR[91,2] = PR[90,2] + -15.063;
   1:  PR[91,3] = PR[90,3] + 30.764;
   1:L PR[91] R[100]mm/sec CNT100;
   1:  PR[91,1] = PR[90,1] + 23.195;
   1:  PR[91,2] = PR[90,2] + -14.857;
   1:  PR[91,3] = PR[90,3] + 30.771;
   1:L PR[91] R[100]mm/sec CNT100;
   1:  PR[91,1] = PR[90,1] + 23.693;
   1:  PR[91,2] = PR[90,2] + -14.540;
   1:  PR[91,3] = PR[90,3] + 30.774;
   1:L PR[91] R[100]mm/sec CNT100;
   1:  PR[91,1] = PR[90,1] + 24.488;
   1:  PR[91,2] = PR[90,2] + -13.978;
   1:  PR[91,3] = PR[90,3] + 30.779;
   1:L PR[91] R[100]mm/sec CNT100;
   1:  PR[91,1] = PR[90,1] + 25.251;
   1:  PR[91,2] = PR[90,2] + -13.381;
   1:  PR[91,3] = PR[90,3] + 30.787;
   1:L PR[91] R[100]mm/sec CNT100;
   1:  PR[91,1] = PR[90,1] + 25.978;
   1:  PR[91,2] = PR[90,2] + -12.749;
   1:  PR[91,3] = PR[90,3] + 30.794;
   1:L PR[91] R[100]mm/sec CNT100;
   1:  PR[91,1] = PR[90,1] + 26.669;
   1:  PR[91,2] = PR[90,2] + -12.083;
   1:  PR[91,3] = PR[90,3] + 30.801;
   1:L PR[91] R[100]mm/sec CNT100;
   1:  PR[91,1] = PR[90,1] + 27.322;
   1:  PR[91,2] = PR[90,2] + -11.384;
   1:  PR[91,3] = PR[90,3] + 30.809;
   1:L PR[91] R[100]mm/sec CNT100;
   1:  PR[91,1] = PR[90,1] + 27.941;
   1:  PR[91,2] = PR[90,2] + -10.650;
   1:  PR[91,3] = PR[90,3] + 30.816;
   1:L PR[91] R[100]mm/sec CNT100;
   1:  PR[91,1] = PR[90,1] + 28.502;
   1:  PR[91,2] = PR[90,2] + -9.913;
   1:  PR[91,3] = PR[90,3] + 30.824;
   1:L PR[91] R[100]mm/sec CNT100;
   1:  PR[91,1] = PR[90,1] + 29.030;
   1:  PR[91,2] = PR[90,2] + -9.141;
   1:  PR[91,3] = PR[90,3] + 30.831;
   1:L PR[91] R[100]mm/sec CNT100;
   1:  PR[91,1] = PR[90,1] + 29.518;
   1:  PR[91,2] = PR[90,2] + -8.345;
   1:  PR[91,3] = PR[90,3] + 30.838;
   1:L PR[91] R[100]mm/sec CNT100;
   1:  PR[91,1] = PR[90,1] + 29.965;
   1:  PR[91,2] = PR[90,2] + -7.531;
   1:  PR[91,3] = PR[90,3] + 30.845;
   1:L PR[91] R[100]mm/sec CNT100;
   1:  PR[91,1] = PR[90,1] + 30.369;
   1:  PR[91,2] = PR[90,2] + -6.702;
   1:  PR[91,3] = PR[90,3] + 30.853;
   1:L PR[91] R[100]mm/sec CNT100;
   1:  PR[91,1] = PR[90,1] + 30.729;
   1:  PR[91,2] = PR[90,2] + -5.864;
   1:  PR[91,3] = PR[90,3] + 30.860;
   1:L PR[91] R[100]mm/sec CNT100;
   1:  PR[91,1] = PR[90,1] + 31.041;
   1:  PR[91,2] = PR[90,2] + -5.018;
   1:  PR[91,3] = PR[90,3] + 30.867;
   1:L PR[91] R[100]mm/sec CNT100;
   1:  PR[91,1] = PR[90,1] + 31.307;
   1:  PR[91,2] = PR[90,2] + -4.163;
   1:  PR[91,3] = PR[90,3] + 30.874;
   1:L PR[91] R[100]mm/sec CNT100;
   1:  PR[91,1] = PR[90,1] + 31.526;
   1:  PR[91,2] = PR[90,2] + -3.294;
   1:  PR[91,3] = PR[90,3] + 30.881;
   1:L PR[91] R[100]mm/sec CNT100;
   1:  PR[91,1] = PR[90,1] + 31.697;
   1:  PR[91,2] = PR[90,2] + -2.407;
   1:  PR[91,3] = PR[90,3] + 30.888;
   1:L PR[91] R[100]mm/sec CNT100;
   1:  PR[91,1] = PR[90,1] + 31.820;
   1:  PR[91,2] = PR[90,2] + -1.495;
   1:  PR[91,3] = PR[90,3] + 30.895;
   1:L PR[91] R[100]mm/sec CNT100;
   1:  PR[91,1] = PR[90,1] + 31.894;
   1:  PR[91,2] = PR[90,2] + -0.552;
   1:  PR[91,3] = PR[90,3] + 30.902;
   1:L PR[91] R[100]mm/sec CNT100;
   1:  PR[91,1] = PR[90,1] + 31.917;
   1:  PR[91,2] = PR[90,2] + 0.428;
   1:  PR[91,3] = PR[90,3] + 30.909;
   1:L PR[91] R[100]mm/sec CNT100;
   1:  PR[91,1] = PR[90,1] + 31.894;
   1:  PR[91,2] = PR[90,2] + 1.408;
   1:  PR[91,3] = PR[90,3] + 30.917;
   1:L PR[91] R[100]mm/sec CNT100;
   1:  PR[91,1] = PR[90,1] + 31.820;
   1:  PR[91,2] = PR[90,2] + 2.350;
   1:  PR[91,3] = PR[90,3] + 30.924;
   1:L PR[91] R[100]mm/sec CNT100;
   1:  PR[91,1] = PR[90,1] + 31.697;
   1:  PR[91,2] = PR[90,2] + 3.262;
   1:  PR[91,3] = PR[90,3] + 30.932;
   1:L PR[91] R[100]mm/sec CNT100;
   1:  PR[91,1] = PR[90,1] + 31.526;
   1:  PR[91,2] = PR[90,2] + 4.150;
   1:  PR[91,3] = PR[90,3] + 30.939;
   1:L PR[91] R[100]mm/sec CNT100;
   1:  PR[91,1] = PR[90,1] + 31.377;
   1:  PR[91,2] = PR[90,2] + 4.748;
   1:  PR[91,3] = PR[90,3] + 30.946;
   1:L PR[91] R[100]mm/sec CNT100;
   1:  PR[91,1] = PR[90,1] + 31.308;
   1:  PR[91,2] = PR[90,2] + 5.017;
   1:  PR[91,3] = PR[90,3] + 30.950;
   1:L PR[91] R[100]mm/sec CNT100;
   1:  PR[91,1] = PR[90,1] + 31.041;
   1:  PR[91,2] = PR[90,2] + 5.873;
   1:  PR[91,3] = PR[90,3] + 30.953;
   1:L PR[91] R[100]mm/sec CNT100;
   1:  PR[91,1] = PR[90,1] + 30.728;
   1:  PR[91,2] = PR[90,2] + 6.719;
   1:  PR[91,3] = PR[90,3] + 30.959;
   1:L PR[91] R[100]mm/sec CNT100;
   1:  PR[91,1] = PR[90,1] + 30.369;
   1:  PR[91,2] = PR[90,2] + 7.558;
   1:  PR[91,3] = PR[90,3] + 30.966;
   1:L PR[91] R[100]mm/sec CNT100;
   1:  PR[91,1] = PR[90,1] + 30.047;
   1:  PR[91,2] = PR[90,2] + 8.221;
   1:  PR[91,3] = PR[90,3] + 30.974;
   1:L PR[91] R[100]mm/sec CNT100;
   1:  PR[91,1] = PR[90,1] + 29.517;
   1:  PR[91,2] = PR[90,2] + 9.202;
   1:  PR[91,3] = PR[90,3] + 30.979;
   1:L PR[91] R[100]mm/sec CNT100;
   1:  PR[91,1] = PR[90,1] + 29.030;
   1:  PR[91,2] = PR[90,2] + 9.996;
   1:  PR[91,3] = PR[90,3] + 30.988;
   1:L PR[91] R[100]mm/sec CNT100;
   1:  PR[91,1] = PR[90,1] + 28.502;
   1:  PR[91,2] = PR[90,2] + 10.768;
   1:  PR[91,3] = PR[90,3] + 30.995;
   1:L PR[91] R[100]mm/sec CNT100;
   1:  PR[91,1] = PR[90,1] + 27.935;
   1:  PR[91,2] = PR[90,2] + 11.512;
   1:  PR[91,3] = PR[90,3] + 31.002;
   1:L PR[91] R[100]mm/sec CNT100;
   1:  PR[91,1] = PR[90,1] + 27.322;
   1:  PR[91,2] = PR[90,2] + 12.239;
   1:  PR[91,3] = PR[90,3] + 31.010;
   1:L PR[91] R[100]mm/sec CNT100;
   1:  PR[91,1] = PR[90,1] + 26.669;
   1:  PR[91,2] = PR[90,2] + 12.938;
   1:  PR[91,3] = PR[90,3] + 31.017;
   1:L PR[91] R[100]mm/sec CNT100;
   1:  PR[91,1] = PR[90,1] + 25.978;
   1:  PR[91,2] = PR[90,2] + 13.604;
   1:  PR[91,3] = PR[90,3] + 31.024;
   1:L PR[91] R[100]mm/sec CNT100;
   1:  PR[91,1] = PR[90,1] + 25.250;
   1:  PR[91,2] = PR[90,2] + 14.236;
   1:  PR[91,3] = PR[90,3] + 31.032;
   1:L PR[91] R[100]mm/sec CNT100;
   1:  PR[91,1] = PR[90,1] + 24.701;
   1:  PR[91,2] = PR[90,2] + 14.668;
   1:  PR[91,3] = PR[90,3] + 31.039;
   1:L PR[91] R[100]mm/sec CNT100;
   1:  PR[91,1] = PR[90,1] + 23.691;
   1:  PR[91,2] = PR[90,2] + 15.396;
   1:  PR[91,3] = PR[90,3] + 31.045;
   1:L PR[91] R[100]mm/sec CNT100;
   1:  PR[91,1] = PR[90,1] + 22.866;
   1:  PR[91,2] = PR[90,2] + 15.919;
   1:  PR[91,3] = PR[90,3] + 31.054;
   1:L PR[91] R[100]mm/sec CNT100;
   1:  PR[91,1] = PR[90,1] + 22.408;
   1:  PR[91,2] = PR[90,2] + 16.181;
   1:  PR[91,3] = PR[90,3] + 31.062;
   1:L PR[91] R[100]mm/sec CNT100;
   1:  PR[91,1] = PR[90,1] + 22.012;
   1:  PR[91,2] = PR[90,2] + 16.403;
   1:  PR[91,3] = PR[90,3] + 31.066;
   1:L PR[91] R[100]mm/sec CNT100;
   1:  PR[91,1] = PR[90,1] + 21.128;
   1:  PR[91,2] = PR[90,2] + 16.848;
   1:  PR[91,3] = PR[90,3] + 31.069;
   1:L PR[91] R[100]mm/sec CNT100;
   1:  PR[91,1] = PR[90,1] + 20.223;
   1:  PR[91,2] = PR[90,2] + 17.250;
   1:  PR[91,3] = PR[90,3] + 31.077;
   1:L PR[91] R[100]mm/sec CNT100;
   1:  PR[91,1] = PR[90,1] + 19.028;
   1:  PR[91,2] = PR[90,2] + 17.700;
   1:  PR[91,3] = PR[90,3] + 31.085;
   1:L PR[91] R[100]mm/sec CNT100;
   1:  PR[91,1] = PR[90,1] + 18.340;
   1:  PR[91,2] = PR[90,2] + 17.927;
   1:  PR[91,3] = PR[90,3] + 31.095;
   1:L PR[91] R[100]mm/sec CNT100;
   1:  PR[91,1] = PR[90,1] + 17.372;
   1:  PR[91,2] = PR[90,2] + 18.196;
   1:  PR[91,3] = PR[90,3] + 31.100;
   1:L PR[91] R[100]mm/sec CNT100;
   1:  PR[91,1] = PR[90,1] + 16.389;
   1:  PR[91,2] = PR[90,2] + 18.418;
   1:  PR[91,3] = PR[90,3] + 31.108;
   1:L PR[91] R[100]mm/sec CNT100;
   1:  PR[91,1] = PR[90,1] + 15.385;
   1:  PR[91,2] = PR[90,2] + 18.593;
   1:  PR[91,3] = PR[90,3] + 31.116;
   1:L PR[91] R[100]mm/sec CNT100;
   1:  PR[91,1] = PR[90,1] + 14.378;
   1:  PR[91,2] = PR[90,2] + 18.720;
   1:  PR[91,3] = PR[90,3] + 31.124;
   1:L PR[91] R[100]mm/sec CNT100;
   1:  PR[91,1] = PR[90,1] + 13.355;
   1:  PR[91,2] = PR[90,2] + 18.797;
   1:  PR[91,3] = PR[90,3] + 31.132;
   1:L PR[91] R[100]mm/sec CNT100;
   1:  PR[91,1] = PR[90,1] + 12.328;
   1:  PR[91,2] = PR[90,2] + 18.823;
   1:  PR[91,3] = PR[90,3] + 31.139;
   1:L PR[91] R[100]mm/sec CNT100;
   1:  PR[91,1] = PR[90,1] + 11.299;
   1:  PR[91,2] = PR[90,2] + 18.797;
   1:  PR[91,3] = PR[90,3] + 31.147;
   1:L PR[91] R[100]mm/sec CNT100;
   1:  PR[91,1] = PR[90,1] + 10.268;
   1:  PR[91,2] = PR[90,2] + 18.719;
   1:  PR[91,3] = PR[90,3] + 31.155;
   1:L PR[91] R[100]mm/sec CNT100;
   1:  PR[91,1] = PR[90,1] + 9.675;
   1:  PR[91,2] = PR[90,2] + 18.649;
   1:  PR[91,3] = PR[90,3] + 31.163;
   1:L PR[91] R[100]mm/sec CNT100;
   1:  PR[91,1] = PR[90,1] + 8.719;
   1:  PR[91,2] = PR[90,2] + 18.500;
   1:  PR[91,3] = PR[90,3] + 31.168;
   1:L PR[91] R[100]mm/sec CNT100;
   1:  PR[91,1] = PR[90,1] + 7.771;
   1:  PR[91,2] = PR[90,2] + 18.306;
   1:  PR[91,3] = PR[90,3] + 31.175;
   1:L PR[91] R[100]mm/sec CNT100;
   1:  PR[91,1] = PR[90,1] + 6.833;
   1:  PR[91,2] = PR[90,2] + 18.067;
   1:  PR[91,3] = PR[90,3] + 31.183;
   1:L PR[91] R[100]mm/sec CNT100;
   1:  PR[91,1] = PR[90,1] + 5.903;
   1:  PR[91,2] = PR[90,2] + 17.781;
   1:  PR[91,3] = PR[90,3] + 31.190;
   1:L PR[91] R[100]mm/sec CNT100;
   1:  PR[91,1] = PR[90,1] + 5.252;
   1:  PR[91,2] = PR[90,2] + 17.552;
   1:  PR[91,3] = PR[90,3] + 31.198;
   1:L PR[91] R[100]mm/sec CNT100;
   1:  PR[91,1] = PR[90,1] + 4.292;
   1:  PR[91,2] = PR[90,2] + 17.166;
   1:  PR[91,3] = PR[90,3] + 31.203;
   1:L PR[91] R[100]mm/sec CNT100;
   1:  PR[91,1] = PR[90,1] + 3.356;
   1:  PR[91,2] = PR[90,2] + 16.732;
   1:  PR[91,3] = PR[90,3] + 31.211;
   1:L PR[91] R[100]mm/sec CNT100;
   1:  PR[91,1] = PR[90,1] + 2.446;
   1:  PR[91,2] = PR[90,2] + 16.251;
   1:  PR[91,3] = PR[90,3] + 31.219;
   1:L PR[91] R[100]mm/sec CNT100;
   1:  PR[91,1] = PR[90,1] + 1.460;
   1:  PR[91,2] = PR[90,2] + 15.658;
   1:  PR[91,3] = PR[90,3] + 31.227;
   1:L PR[91] R[100]mm/sec CNT100;
   1:  PR[91,1] = PR[90,1] + 1.102;
   1:  PR[91,2] = PR[90,2] + 15.462;
   1:  PR[91,3] = PR[90,3] + 31.236;
   1:L PR[91] R[100]mm/sec CNT100;
   1:  PR[91,1] = PR[90,1] + 0.635;
   1:  PR[91,2] = PR[90,2] + 15.292;
   1:  PR[91,3] = PR[90,3] + 31.239;
   1:L PR[91] R[100]mm/sec CNT100;
   1:  PR[91,1] = PR[90,1] + 0.148;
   1:  PR[91,2] = PR[90,2] + 15.208;
   1:  PR[91,3] = PR[90,3] + 31.243;
   1:L PR[91] R[100]mm/sec CNT100;
   1:  PR[91,1] = PR[90,1] + -0.344;
   1:  PR[91,2] = PR[90,2] + 15.201;
   1:  PR[91,3] = PR[90,3] + 31.247;
   1:L PR[91] R[100]mm/sec CNT100;
   1:  PR[91,1] = PR[90,1] + -0.831;
   1:  PR[91,2] = PR[90,2] + 15.281;
   1:  PR[91,3] = PR[90,3] + 31.251;
   1:L PR[91] R[100]mm/sec CNT100;
   1:  PR[91,1] = PR[90,1] + -1.298;
   1:  PR[91,2] = PR[90,2] + 15.438;
   1:  PR[91,3] = PR[90,3] + 31.255;
   1:L PR[91] R[100]mm/sec CNT100;
   1:  PR[91,1] = PR[90,1] + -1.702;
   1:  PR[91,2] = PR[90,2] + 15.657;
   1:  PR[91,3] = PR[90,3] + 31.258;
   1:L PR[91] R[100]mm/sec CNT100;
   1:  PR[91,1] = PR[90,1] + -2.690;
   1:  PR[91,2] = PR[90,2] + 16.252;
   1:  PR[91,3] = PR[90,3] + 31.262;
   1:L PR[91] R[100]mm/sec CNT100;
   1:  PR[91,1] = PR[90,1] + -3.456;
   1:  PR[91,2] = PR[90,2] + 16.662;
   1:  PR[91,3] = PR[90,3] + 31.271;
   1:L PR[91] R[100]mm/sec CNT100;
   1:  PR[91,1] = PR[90,1] + -4.336;
   1:  PR[91,2] = PR[90,2] + 17.080;
   1:  PR[91,3] = PR[90,3] + 31.278;
   1:L PR[91] R[100]mm/sec CNT100;
   1:  PR[91,1] = PR[90,1] + -5.232;
   1:  PR[91,2] = PR[90,2] + 17.454;
   1:  PR[91,3] = PR[90,3] + 31.285;
   1:L PR[91] R[100]mm/sec CNT100;
   1:  PR[91,1] = PR[90,1] + -6.473;
   1:  PR[91,2] = PR[90,2] + 17.891;
   1:  PR[91,3] = PR[90,3] + 31.293;
   1:L PR[91] R[100]mm/sec CNT100;
   1:  PR[91,1] = PR[90,1] + -7.467;
   1:  PR[91,2] = PR[90,2] + 18.176;
   1:  PR[91,3] = PR[90,3] + 31.303;
   1:L PR[91] R[100]mm/sec CNT100;
   1:  PR[91,1] = PR[90,1] + -8.010;
   1:  PR[91,2] = PR[90,2] + 18.308;
   1:  PR[91,3] = PR[90,3] + 31.311;
   1:L PR[91] R[100]mm/sec CNT100;
   1:  PR[91,1] = PR[90,1] + -8.960;
   1:  PR[91,2] = PR[90,2] + 18.501;
   1:  PR[91,3] = PR[90,3] + 31.315;
   1:L PR[91] R[100]mm/sec CNT100;
   1:  PR[91,1] = PR[90,1] + -9.914;
   1:  PR[91,2] = PR[90,2] + 18.649;
   1:  PR[91,3] = PR[90,3] + 31.323;
   1:L PR[91] R[100]mm/sec CNT100;
   1:  PR[91,1] = PR[90,1] + -10.871;
   1:  PR[91,2] = PR[90,2] + 18.751;
   1:  PR[91,3] = PR[90,3] + 31.330;
   1:L PR[91] R[100]mm/sec CNT100;
   1:  PR[91,1] = PR[90,1] + -11.832;
   1:  PR[91,2] = PR[90,2] + 18.808;
   1:  PR[91,3] = PR[90,3] + 31.338;
   1:L PR[91] R[100]mm/sec CNT100;
   1:  PR[91,1] = PR[90,1] + -12.568;
   1:  PR[91,2] = PR[90,2] + 18.823;
   1:  PR[91,3] = PR[90,3] + 31.345;
   1:L PR[91] R[100]mm/sec CNT100;
   1:  PR[91,1] = PR[90,1] + -13.597;
   1:  PR[91,2] = PR[90,2] + 18.796;
   1:  PR[91,3] = PR[90,3] + 31.351;
   1:L PR[91] R[100]mm/sec CNT100;
   1:  PR[91,1] = PR[90,1] + -14.619;
   1:  PR[91,2] = PR[90,2] + 18.719;
   1:  PR[91,3] = PR[90,3] + 31.359;
   1:L PR[91] R[100]mm/sec CNT100;
   1:  PR[91,1] = PR[90,1] + -15.634;
   1:  PR[91,2] = PR[90,2] + 18.591;
   1:  PR[91,3] = PR[90,3] + 31.367;
   1:L PR[91] R[100]mm/sec CNT100;
   1:  PR[91,1] = PR[90,1] + -16.587;
   1:  PR[91,2] = PR[90,2] + 18.426;
   1:  PR[91,3] = PR[90,3] + 31.375;
   1:L PR[91] R[100]mm/sec CNT100;
   1:  PR[91,1] = PR[90,1] + -17.533;
   1:  PR[91,2] = PR[90,2] + 18.216;
   1:  PR[91,3] = PR[90,3] + 31.382;
   1:L PR[91] R[100]mm/sec CNT100;
   1:  PR[91,1] = PR[90,1] + -18.465;
   1:  PR[91,2] = PR[90,2] + 17.962;
   1:  PR[91,3] = PR[90,3] + 31.390;
   1:L PR[91] R[100]mm/sec CNT100;
   1:  PR[91,1] = PR[90,1] + -19.670;
   1:  PR[91,2] = PR[90,2] + 17.560;
   1:  PR[91,3] = PR[90,3] + 31.397;
   1:L PR[91] R[100]mm/sec CNT100;
   1:  PR[91,1] = PR[90,1] + -20.636;
   1:  PR[91,2] = PR[90,2] + 17.176;
   1:  PR[91,3] = PR[90,3] + 31.407;
   1:L PR[91] R[100]mm/sec CNT100;
   1:  PR[91,1] = PR[90,1] + -21.586;
   1:  PR[91,2] = PR[90,2] + 16.740;
   1:  PR[91,3] = PR[90,3] + 31.415;
   1:L PR[91] R[100]mm/sec CNT100;
   1:  PR[91,1] = PR[90,1] + -22.047;
   1:  PR[91,2] = PR[90,2] + 16.509;
   1:  PR[91,3] = PR[90,3] + 31.423;
   1:L PR[91] R[100]mm/sec CNT100;
   1:  PR[91,1] = PR[90,1] + -22.895;
   1:  PR[91,2] = PR[90,2] + 16.041;
   1:  PR[91,3] = PR[90,3] + 31.427;
   1:L PR[91] R[100]mm/sec CNT100;
   1:  PR[91,1] = PR[90,1] + -23.716;
   1:  PR[91,2] = PR[90,2] + 15.534;
   1:  PR[91,3] = PR[90,3] + 31.435;
   1:L PR[91] R[100]mm/sec CNT100;
   1:  PR[91,1] = PR[90,1] + -24.510;
   1:  PR[91,2] = PR[90,2] + 14.989;
   1:  PR[91,3] = PR[90,3] + 31.442;
   1:L PR[91] R[100]mm/sec CNT100;
   1:  PR[91,1] = PR[90,1] + -25.275;
   1:  PR[91,2] = PR[90,2] + 14.406;
   1:  PR[91,3] = PR[90,3] + 31.449;
   1:L PR[91] R[100]mm/sec CNT100;
   1:  PR[91,1] = PR[90,1] + -25.869;
   1:  PR[91,2] = PR[90,2] + 13.909;
   1:  PR[91,3] = PR[90,3] + 31.457;
   1:L PR[91] R[100]mm/sec CNT100;
   1:  PR[91,1] = PR[90,1] + -26.710;
   1:  PR[91,2] = PR[90,2] + 13.135;
   1:  PR[91,3] = PR[90,3] + 31.463;
   1:L PR[91] R[100]mm/sec CNT100;
   1:  PR[91,1] = PR[90,1] + -27.374;
   1:  PR[91,2] = PR[90,2] + 12.449;
   1:  PR[91,3] = PR[90,3] + 31.472;
   1:L PR[91] R[100]mm/sec CNT100;
   1:  PR[91,1] = PR[90,1] + -28.003;
   1:  PR[91,2] = PR[90,2] + 11.728;
   1:  PR[91,3] = PR[90,3] + 31.479;
   1:L PR[91] R[100]mm/sec CNT100;
   1:  PR[91,1] = PR[90,1] + -28.600;
   1:  PR[91,2] = PR[90,2] + 10.969;
   1:  PR[91,3] = PR[90,3] + 31.487;
   1:L PR[91] R[100]mm/sec CNT100;
   1:  PR[91,1] = PR[90,1] + -29.155;
   1:  PR[91,2] = PR[90,2] + 10.179;
   1:  PR[91,3] = PR[90,3] + 31.494;
   1:L PR[91] R[100]mm/sec CNT100;
   1:  PR[91,1] = PR[90,1] + -29.666;
   1:  PR[91,2] = PR[90,2] + 9.364;
   1:  PR[91,3] = PR[90,3] + 31.501;
   1:L PR[91] R[100]mm/sec CNT100;
   1:  PR[91,1] = PR[90,1] + -30.133;
   1:  PR[91,2] = PR[90,2] + 8.526;
   1:  PR[91,3] = PR[90,3] + 31.509;
   1:L PR[91] R[100]mm/sec CNT100;
   1:  PR[91,1] = PR[90,1] + -30.553;
   1:  PR[91,2] = PR[90,2] + 7.673;
   1:  PR[91,3] = PR[90,3] + 31.516;
   1:L PR[91] R[100]mm/sec CNT100;
   1:  PR[91,1] = PR[90,1] + -30.927;
   1:  PR[91,2] = PR[90,2] + 6.809;
   1:  PR[91,3] = PR[90,3] + 31.524;
   1:L PR[91] R[100]mm/sec CNT100;
   1:  PR[91,1] = PR[90,1] + -31.252;
   1:  PR[91,2] = PR[90,2] + 5.940;
   1:  PR[91,3] = PR[90,3] + 31.531;
   1:L PR[91] R[100]mm/sec CNT100;
   1:  PR[91,1] = PR[90,1] + -31.527;
   1:  PR[91,2] = PR[90,2] + 5.066;
   1:  PR[91,3] = PR[90,3] + 31.538;
   1:L PR[91] R[100]mm/sec CNT100;
   1:  PR[91,1] = PR[90,1] + -31.753;
   1:  PR[91,2] = PR[90,2] + 4.185;
   1:  PR[91,3] = PR[90,3] + 31.545;
   1:L PR[91] R[100]mm/sec CNT100;
   1:  PR[91,1] = PR[90,1] + -31.929;
   1:  PR[91,2] = PR[90,2] + 3.289;
   1:  PR[91,3] = PR[90,3] + 31.552;
   1:L PR[91] R[100]mm/sec CNT100;
   1:  PR[91,1] = PR[90,1] + -32.055;
   1:  PR[91,2] = PR[90,2] + 2.370;
   1:  PR[91,3] = PR[90,3] + 31.559;
   1:L PR[91] R[100]mm/sec CNT100;
   1:  PR[91,1] = PR[90,1] + -32.132;
   1:  PR[91,2] = PR[90,2] + 1.419;
   1:  PR[91,3] = PR[90,3] + 31.567;
   1:L PR[91] R[100]mm/sec CNT100;
   1:  PR[91,1] = PR[90,1] + -32.155;
   1:  PR[91,2] = PR[90,2] + 0.428;
   1:  PR[91,3] = PR[90,3] + 31.574;
   1:L PR[91] R[100]mm/sec CNT100;
   1:  PR[91,1] = PR[90,1] + -32.132;
   1:  PR[91,2] = PR[90,2] + -0.564;
   1:  PR[91,3] = PR[90,3] + 31.582;
   1:L PR[91] R[100]mm/sec CNT100;
   1:  PR[91,1] = PR[90,1] + -32.055;
   1:  PR[91,2] = PR[90,2] + -1.515;
   1:  PR[91,3] = PR[90,3] + 31.589;
   1:L PR[91] R[100]mm/sec CNT100;
   1:  PR[91,1] = PR[90,1] + -31.929;
   1:  PR[91,2] = PR[90,2] + -2.434;
   1:  PR[91,3] = PR[90,3] + 31.597;
   1:L PR[91] R[100]mm/sec CNT100;
   1:  PR[91,1] = PR[90,1] + -31.753;
   1:  PR[91,2] = PR[90,2] + -3.329;
   1:  PR[91,3] = PR[90,3] + 31.604;
   1:L PR[91] R[100]mm/sec CNT100;
   1:  PR[91,1] = PR[90,1] + -31.527;
   1:  PR[91,2] = PR[90,2] + -4.211;
   1:  PR[91,3] = PR[90,3] + 31.611;
   1:L PR[91] R[100]mm/sec CNT100;
   1:  PR[91,1] = PR[90,1] + -31.252;
   1:  PR[91,2] = PR[90,2] + -5.085;
   1:  PR[91,3] = PR[90,3] + 31.618;
   1:L PR[91] R[100]mm/sec CNT100;
   1:  PR[91,1] = PR[90,1] + -30.927;
   1:  PR[91,2] = PR[90,2] + -5.954;
   1:  PR[91,3] = PR[90,3] + 31.625;
   1:L PR[91] R[100]mm/sec CNT100;
   1:  PR[91,1] = PR[90,1] + -30.553;
   1:  PR[91,2] = PR[90,2] + -6.817;
   1:  PR[91,3] = PR[90,3] + 31.632;
   1:L PR[91] R[100]mm/sec CNT100;
   1:  PR[91,1] = PR[90,1] + -30.133;
   1:  PR[91,2] = PR[90,2] + -7.671;
   1:  PR[91,3] = PR[90,3] + 31.640;
   1:L PR[91] R[100]mm/sec CNT100;
   1:  PR[91,1] = PR[90,1] + -29.666;
   1:  PR[91,2] = PR[90,2] + -8.509;
   1:  PR[91,3] = PR[90,3] + 31.647;
   1:L PR[91] R[100]mm/sec CNT100;
   1:  PR[91,1] = PR[90,1] + -29.155;
   1:  PR[91,2] = PR[90,2] + -9.324;
   1:  PR[91,3] = PR[90,3] + 31.654;
   1:L PR[91] R[100]mm/sec CNT100;
   1:  PR[91,1] = PR[90,1] + -28.600;
   1:  PR[91,2] = PR[90,2] + -10.114;
   1:  PR[91,3] = PR[90,3] + 31.662;
   1:L PR[91] R[100]mm/sec CNT100;
   1:  PR[91,1] = PR[90,1] + -27.999;
   1:  PR[91,2] = PR[90,2] + -10.878;
   1:  PR[91,3] = PR[90,3] + 31.669;
   1:L PR[91] R[100]mm/sec CNT100;
   1:  PR[91,1] = PR[90,1] + -27.375;
   1:  PR[91,2] = PR[90,2] + -11.593;
   1:  PR[91,3] = PR[90,3] + 31.677;
   1:L PR[91] R[100]mm/sec CNT100;
   1:  PR[91,1] = PR[90,1] + -26.622;
   1:  PR[91,2] = PR[90,2] + -12.363;
   1:  PR[91,3] = PR[90,3] + 31.684;
   1:L PR[91] R[100]mm/sec CNT100;
   1:  PR[91,1] = PR[90,1] + -25.870;
   1:  PR[91,2] = PR[90,2] + -13.053;
   1:  PR[91,3] = PR[90,3] + 31.692;
   1:L PR[91] R[100]mm/sec CNT100;
   1:  PR[91,1] = PR[90,1] + -25.275;
   1:  PR[91,2] = PR[90,2] + -13.551;
   1:  PR[91,3] = PR[90,3] + 31.700;
   1:L PR[91] R[100]mm/sec CNT100;
   1:  PR[91,1] = PR[90,1] + -24.510;
   1:  PR[91,2] = PR[90,2] + -14.134;
   1:  PR[91,3] = PR[90,3] + 31.706;
   1:L PR[91] R[100]mm/sec CNT100;
   1:  PR[91,1] = PR[90,1] + -23.716;
   1:  PR[91,2] = PR[90,2] + -14.679;
   1:  PR[91,3] = PR[90,3] + 31.714;
   1:L PR[91] R[100]mm/sec CNT100;
   1:  PR[91,1] = PR[90,1] + -22.895;
   1:  PR[91,2] = PR[90,2] + -15.185;
   1:  PR[91,3] = PR[90,3] + 31.721;
   1:L PR[91] R[100]mm/sec CNT100;
   1:  PR[91,1] = PR[90,1] + -22.049;
   1:  PR[91,2] = PR[90,2] + -15.653;
   1:  PR[91,3] = PR[90,3] + 31.729;
   1:L PR[91] R[100]mm/sec CNT100;
   1:  PR[91,1] = PR[90,1] + -21.180;
   1:  PR[91,2] = PR[90,2] + -16.081;
   1:  PR[91,3] = PR[90,3] + 31.736;
   1:L PR[91] R[100]mm/sec CNT100;
   1:  PR[91,1] = PR[90,1] + -20.641;
   1:  PR[91,2] = PR[90,2] + -16.319;
   1:  PR[91,3] = PR[90,3] + 31.744;
   1:L PR[91] R[100]mm/sec CNT100;
   1:  PR[91,1] = PR[90,1] + -19.669;
   1:  PR[91,2] = PR[90,2] + -16.705;
   1:  PR[91,3] = PR[90,3] + 31.748;
   1:L PR[91] R[100]mm/sec CNT100;
   1:  PR[91,1] = PR[90,1] + -18.683;
   1:  PR[91,2] = PR[90,2] + -17.040;
   1:  PR[91,3] = PR[90,3] + 31.756;
   1:L PR[91] R[100]mm/sec CNT100;
   1:  PR[91,1] = PR[90,1] + -17.531;
   1:  PR[91,2] = PR[90,2] + -17.361;
   1:  PR[91,3] = PR[90,3] + 31.764;
   1:L PR[91] R[100]mm/sec CNT100;
   1:  PR[91,1] = PR[90,1] + -16.663;
   1:  PR[91,2] = PR[90,2] + -17.556;
   1:  PR[91,3] = PR[90,3] + 31.774;
   1:L PR[91] R[100]mm/sec CNT100;
   1:  PR[91,1] = PR[90,1] + -15.624;
   1:  PR[91,2] = PR[90,2] + -17.738;
   1:  PR[91,3] = PR[90,3] + 31.780;
   1:L PR[91] R[100]mm/sec CNT100;
   1:  PR[91,1] = PR[90,1] + -14.620;
   1:  PR[91,2] = PR[90,2] + -17.864;
   1:  PR[91,3] = PR[90,3] + 31.789;
   1:L PR[91] R[100]mm/sec CNT100;
   1:  PR[91,1] = PR[90,1] + -13.597;
   1:  PR[91,2] = PR[90,2] + -17.941;
   1:  PR[91,3] = PR[90,3] + 31.796;
   1:L PR[91] R[100]mm/sec CNT100;
   1:  PR[91,1] = PR[90,1] + -12.570;
   1:  PR[91,2] = PR[90,2] + -17.967;
   1:  PR[91,3] = PR[90,3] + 31.804;
   1:L PR[91] R[100]mm/sec CNT100;
   1:  PR[91,1] = PR[90,1] + -11.541;
   1:  PR[91,2] = PR[90,2] + -17.942;
   1:  PR[91,3] = PR[90,3] + 31.812;
   1:L PR[91] R[100]mm/sec CNT100;
   1:  PR[91,1] = PR[90,1] + -10.513;
   1:  PR[91,2] = PR[90,2] + -17.864;
   1:  PR[91,3] = PR[90,3] + 31.820;
   1:L PR[91] R[100]mm/sec CNT100;
   1:  PR[91,1] = PR[90,1] + -9.488;
   1:  PR[91,2] = PR[90,2] + -17.735;
   1:  PR[91,3] = PR[90,3] + 31.828;
   1:L PR[91] R[100]mm/sec CNT100;
   1:  PR[91,1] = PR[90,1] + -8.471;
   1:  PR[91,2] = PR[90,2] + -17.554;
   1:  PR[91,3] = PR[90,3] + 31.836;
   1:L PR[91] R[100]mm/sec CNT100;
   1:  PR[91,1] = PR[90,1] + -7.460;
   1:  PR[91,2] = PR[90,2] + -17.319;
   1:  PR[91,3] = PR[90,3] + 31.844;
   1:L PR[91] R[100]mm/sec CNT100;
   1:  PR[91,1] = PR[90,1] + -7.080;
   1:  PR[91,2] = PR[90,2] + -17.216;
   1:  PR[91,3] = PR[90,3] + 31.852;
   1:L PR[91] R[100]mm/sec CNT100;
   1:  PR[91,1] = PR[90,1] + -6.148;
   1:  PR[91,2] = PR[90,2] + -16.930;
   1:  PR[91,3] = PR[90,3] + 31.855;
   1:L PR[91] R[100]mm/sec CNT100;
   1:  PR[91,1] = PR[90,1] + -5.234;
   1:  PR[91,2] = PR[90,2] + -16.600;
   1:  PR[91,3] = PR[90,3] + 31.863;
   1:L PR[91] R[100]mm/sec CNT100;
   1:  PR[91,1] = PR[90,1] + -4.336;
   1:  PR[91,2] = PR[90,2] + -16.225;
   1:  PR[91,3] = PR[90,3] + 31.870;
   1:L PR[91] R[100]mm/sec CNT100;
   1:  PR[91,1] = PR[90,1] + -3.456;
   1:  PR[91,2] = PR[90,2] + -15.806;
   1:  PR[91,3] = PR[90,3] + 31.878;
   1:L PR[91] R[100]mm/sec CNT100;
   1:  PR[91,1] = PR[90,1] + -2.690;
   1:  PR[91,2] = PR[90,2] + -15.397;
   1:  PR[91,3] = PR[90,3] + 31.886;
   1:L PR[91] R[100]mm/sec CNT100;
   1:  PR[91,1] = PR[90,1] + -1.703;
   1:  PR[91,2] = PR[90,2] + -14.802;
   1:  PR[91,3] = PR[90,3] + 31.892;
   1:L PR[91] R[100]mm/sec CNT100;
   1:  PR[91,1] = PR[90,1] + -1.298;
   1:  PR[91,2] = PR[90,2] + -14.583;
   1:  PR[91,3] = PR[90,3] + 31.901;
   1:L PR[91] R[100]mm/sec CNT100;
   1:  PR[91,1] = PR[90,1] + -0.831;
   1:  PR[91,2] = PR[90,2] + -14.425;
   1:  PR[91,3] = PR[90,3] + 31.905;
   1:L PR[91] R[100]mm/sec CNT100;
   1:  PR[91,1] = PR[90,1] + -0.344;
   1:  PR[91,2] = PR[90,2] + -14.346;
   1:  PR[91,3] = PR[90,3] + 31.909;
   1:L PR[91] R[100]mm/sec CNT100;
   1:  PR[91,1] = PR[90,1] + 0.148;
   1:  PR[91,2] = PR[90,2] + -14.353;
   1:  PR[91,3] = PR[90,3] + 31.912;
   1:L PR[91] R[100]mm/sec CNT100;
   1:  PR[91,1] = PR[90,1] + 0.635;
   1:  PR[91,2] = PR[90,2] + -14.437;
   1:  PR[91,3] = PR[90,3] + 31.916;
   1:L PR[91] R[100]mm/sec CNT100;
   1:  PR[91] = PR[90];
   1:  PR[91,1] = PR[90,1] + 0.721;
   1:  PR[91,2] = PR[90,2] + -14.967;
   1:  PR[91,3] = PR[90,3] + 33.250;
   1:L PR[91] R[100]mm/sec CNT100;
   1:  PR[91,1] = PR[90,1] + 1.180;
   1:  PR[91,2] = PR[90,2] + -15.147;
   1:  PR[91,3] = PR[90,3] + 31.923;
   1:L PR[91] R[100]mm/sec CNT100;
   1:  PR[91,1] = PR[90,1] + 1.934;
   1:  PR[91,2] = PR[90,2] + -15.581;
   1:  PR[91,3] = PR[90,3] + 31.926;
   1:L PR[91] R[100]mm/sec CNT100;
   1:  PR[91,1] = PR[90,1] + 2.539;
   1:  PR[91,2] = PR[90,2] + -15.902;
   1:  PR[91,3] = PR[90,3] + 31.933;
   1:L PR[91] R[100]mm/sec CNT100;
   1:  PR[91,1] = PR[90,1] + 3.486;
   1:  PR[91,2] = PR[90,2] + -16.355;
   1:  PR[91,3] = PR[90,3] + 31.939;
   1:L PR[91] R[100]mm/sec CNT100;
   1:  PR[91,1] = PR[90,1] + 4.631;
   1:  PR[91,2] = PR[90,2] + -16.826;
   1:  PR[91,3] = PR[90,3] + 31.947;
   1:L PR[91] R[100]mm/sec CNT100;
   1:  PR[91,1] = PR[90,1] + 5.450;
   1:  PR[91,2] = PR[90,2] + -17.112;
   1:  PR[91,3] = PR[90,3] + 31.956;
   1:L PR[91] R[100]mm/sec CNT100;
   1:  PR[91,1] = PR[90,1] + 6.522;
   1:  PR[91,2] = PR[90,2] + -17.430;
   1:  PR[91,3] = PR[90,3] + 31.963;
   1:L PR[91] R[100]mm/sec CNT100;
   1:  PR[91,1] = PR[90,1] + 7.497;
   1:  PR[91,2] = PR[90,2] + -17.665;
   1:  PR[91,3] = PR[90,3] + 31.972;
   1:L PR[91] R[100]mm/sec CNT100;
   1:  PR[91,1] = PR[90,1] + 8.448;
   1:  PR[91,2] = PR[90,2] + -17.846;
   1:  PR[91,3] = PR[90,3] + 31.980;
   1:L PR[91] R[100]mm/sec CNT100;
   1:  PR[91,1] = PR[90,1] + 9.559;
   1:  PR[91,2] = PR[90,2] + -17.999;
   1:  PR[91,3] = PR[90,3] + 31.987;
   1:L PR[91] R[100]mm/sec CNT100;
   1:  PR[91,1] = PR[90,1] + 10.387;
   1:  PR[91,2] = PR[90,2] + -18.073;
   1:  PR[91,3] = PR[90,3] + 31.996;
   1:L PR[91] R[100]mm/sec CNT100;
   1:  PR[91,1] = PR[90,1] + 11.360;
   1:  PR[91,2] = PR[90,2] + -18.116;
   1:  PR[91,3] = PR[90,3] + 32.003;
   1:L PR[91] R[100]mm/sec CNT100;
   1:  PR[91,1] = PR[90,1] + 12.337;
   1:  PR[91,2] = PR[90,2] + -18.114;
   1:  PR[91,3] = PR[90,3] + 32.010;
   1:L PR[91] R[100]mm/sec CNT100;
   1:  PR[91,1] = PR[90,1] + 12.671;
   1:  PR[91,2] = PR[90,2] + -18.104;
   1:  PR[91,3] = PR[90,3] + 32.018;
   1:L PR[91] R[100]mm/sec CNT100;
   1:  PR[91,1] = PR[90,1] + 13.709;
   1:  PR[91,2] = PR[90,2] + -18.034;
   1:  PR[91,3] = PR[90,3] + 32.020;
   1:L PR[91] R[100]mm/sec CNT100;
   1:  PR[91,1] = PR[90,1] + 14.735;
   1:  PR[91,2] = PR[90,2] + -17.913;
   1:  PR[91,3] = PR[90,3] + 32.029;
   1:L PR[91] R[100]mm/sec CNT100;
   1:  PR[91,1] = PR[90,1] + 15.751;
   1:  PR[91,2] = PR[90,2] + -17.741;
   1:  PR[91,3] = PR[90,3] + 32.037;
   1:L PR[91] R[100]mm/sec CNT100;
   1:  PR[91,1] = PR[90,1] + 16.754;
   1:  PR[91,2] = PR[90,2] + -17.519;
   1:  PR[91,3] = PR[90,3] + 32.045;
   1:L PR[91] R[100]mm/sec CNT100;
   1:  PR[91,1] = PR[90,1] + 17.739;
   1:  PR[91,2] = PR[90,2] + -17.248;
   1:  PR[91,3] = PR[90,3] + 32.053;
   1:L PR[91] R[100]mm/sec CNT100;
   1:  PR[91,1] = PR[90,1] + 18.898;
   1:  PR[91,2] = PR[90,2] + -16.859;
   1:  PR[91,3] = PR[90,3] + 32.061;
   1:L PR[91] R[100]mm/sec CNT100;
   1:  PR[91,1] = PR[90,1] + 19.656;
   1:  PR[91,2] = PR[90,2] + -16.566;
   1:  PR[91,3] = PR[90,3] + 32.070;
   1:L PR[91] R[100]mm/sec CNT100;
   1:  PR[91,1] = PR[90,1] + 20.580;
   1:  PR[91,2] = PR[90,2] + -16.157;
   1:  PR[91,3] = PR[90,3] + 32.077;
   1:L PR[91] R[100]mm/sec CNT100;
   1:  PR[91,1] = PR[90,1] + 21.478;
   1:  PR[91,2] = PR[90,2] + -15.707;
   1:  PR[91,3] = PR[90,3] + 32.085;
   1:L PR[91] R[100]mm/sec CNT100;
   1:  PR[91,1] = PR[90,1] + 22.344;
   1:  PR[91,2] = PR[90,2] + -15.219;
   1:  PR[91,3] = PR[90,3] + 32.092;
   1:L PR[91] R[100]mm/sec CNT100;
   1:  PR[91,1] = PR[90,1] + 23.180;
   1:  PR[91,2] = PR[90,2] + -14.693;
   1:  PR[91,3] = PR[90,3] + 32.100;
   1:L PR[91] R[100]mm/sec CNT100;
   1:  PR[91,1] = PR[90,1] + 23.985;
   1:  PR[91,2] = PR[90,2] + -14.128;
   1:  PR[91,3] = PR[90,3] + 32.108;
   1:L PR[91] R[100]mm/sec CNT100;
   1:  PR[91,1] = PR[90,1] + 24.756;
   1:  PR[91,2] = PR[90,2] + -13.526;
   1:  PR[91,3] = PR[90,3] + 32.116;
   1:L PR[91] R[100]mm/sec CNT100;
   1:  PR[91,1] = PR[90,1] + 25.492;
   1:  PR[91,2] = PR[90,2] + -12.889;
   1:  PR[91,3] = PR[90,3] + 32.123;
   1:L PR[91] R[100]mm/sec CNT100;
   1:  PR[91,1] = PR[90,1] + 26.192;
   1:  PR[91,2] = PR[90,2] + -12.218;
   1:  PR[91,3] = PR[90,3] + 32.131;
   1:L PR[91] R[100]mm/sec CNT100;
   1:  PR[91,1] = PR[90,1] + 26.854;
   1:  PR[91,2] = PR[90,2] + -11.514;
   1:  PR[91,3] = PR[90,3] + 32.138;
   1:L PR[91] R[100]mm/sec CNT100;
   1:  PR[91,1] = PR[90,1] + 27.476;
   1:  PR[91,2] = PR[90,2] + -10.779;
   1:  PR[91,3] = PR[90,3] + 32.146;
   1:L PR[91] R[100]mm/sec CNT100;
   1:  PR[91,1] = PR[90,1] + 28.057;
   1:  PR[91,2] = PR[90,2] + -10.015;
   1:  PR[91,3] = PR[90,3] + 32.153;
   1:L PR[91] R[100]mm/sec CNT100;
   1:  PR[91,1] = PR[90,1] + 28.596;
   1:  PR[91,2] = PR[90,2] + -9.225;
   1:  PR[91,3] = PR[90,3] + 32.161;
   1:L PR[91] R[100]mm/sec CNT100;
   1:  PR[91,1] = PR[90,1] + 29.092;
   1:  PR[91,2] = PR[90,2] + -8.413;
   1:  PR[91,3] = PR[90,3] + 32.168;
   1:L PR[91] R[100]mm/sec CNT100;
   1:  PR[91,1] = PR[90,1] + 29.545;
   1:  PR[91,2] = PR[90,2] + -7.584;
   1:  PR[91,3] = PR[90,3] + 32.176;
   1:L PR[91] R[100]mm/sec CNT100;
   1:  PR[91,1] = PR[90,1] + 29.952;
   1:  PR[91,2] = PR[90,2] + -6.743;
   1:  PR[91,3] = PR[90,3] + 32.183;
   1:L PR[91] R[100]mm/sec CNT100;
   1:  PR[91,1] = PR[90,1] + 30.313;
   1:  PR[91,2] = PR[90,2] + -5.895;
   1:  PR[91,3] = PR[90,3] + 32.191;
   1:L PR[91] R[100]mm/sec CNT100;
   1:  PR[91,1] = PR[90,1] + 30.627;
   1:  PR[91,2] = PR[90,2] + -5.040;
   1:  PR[91,3] = PR[90,3] + 32.198;
   1:L PR[91] R[100]mm/sec CNT100;
   1:  PR[91,1] = PR[90,1] + 30.893;
   1:  PR[91,2] = PR[90,2] + -4.178;
   1:  PR[91,3] = PR[90,3] + 32.205;
   1:L PR[91] R[100]mm/sec CNT100;
   1:  PR[91,1] = PR[90,1] + 31.111;
   1:  PR[91,2] = PR[90,2] + -3.303;
   1:  PR[91,3] = PR[90,3] + 32.212;
   1:L PR[91] R[100]mm/sec CNT100;
   1:  PR[91,1] = PR[90,1] + 31.281;
   1:  PR[91,2] = PR[90,2] + -2.411;
   1:  PR[91,3] = PR[90,3] + 32.219;
   1:L PR[91] R[100]mm/sec CNT100;
   1:  PR[91,1] = PR[90,1] + 31.403;
   1:  PR[91,2] = PR[90,2] + -1.496;
   1:  PR[91,3] = PR[90,3] + 32.226;
   1:L PR[91] R[100]mm/sec CNT100;
   1:  PR[91,1] = PR[90,1] + 31.476;
   1:  PR[91,2] = PR[90,2] + -0.552;
   1:  PR[91,3] = PR[90,3] + 32.233;
   1:L PR[91] R[100]mm/sec CNT100;
   1:  PR[91,1] = PR[90,1] + 31.501;
   1:  PR[91,2] = PR[90,2] + 0.428;
   1:  PR[91,3] = PR[90,3] + 32.241;
   1:L PR[91] R[100]mm/sec CNT100;
   1:  PR[91,1] = PR[90,1] + 31.476;
   1:  PR[91,2] = PR[90,2] + 1.407;
   1:  PR[91,3] = PR[90,3] + 32.248;
   1:L PR[91] R[100]mm/sec CNT100;
   1:  PR[91,1] = PR[90,1] + 31.403;
   1:  PR[91,2] = PR[90,2] + 2.352;
   1:  PR[91,3] = PR[90,3] + 32.256;
   1:L PR[91] R[100]mm/sec CNT100;
   1:  PR[91,1] = PR[90,1] + 31.281;
   1:  PR[91,2] = PR[90,2] + 3.267;
   1:  PR[91,3] = PR[90,3] + 32.263;
   1:L PR[91] R[100]mm/sec CNT100;
   1:  PR[91,1] = PR[90,1] + 31.111;
   1:  PR[91,2] = PR[90,2] + 4.158;
   1:  PR[91,3] = PR[90,3] + 32.271;
   1:L PR[91] R[100]mm/sec CNT100;
   1:  PR[91,1] = PR[90,1] + 30.893;
   1:  PR[91,2] = PR[90,2] + 5.033;
   1:  PR[91,3] = PR[90,3] + 32.278;
   1:L PR[91] R[100]mm/sec CNT100;
   1:  PR[91,1] = PR[90,1] + 30.627;
   1:  PR[91,2] = PR[90,2] + 5.895;
   1:  PR[91,3] = PR[90,3] + 32.285;
   1:L PR[91] R[100]mm/sec CNT100;
   1:  PR[91,1] = PR[90,1] + 30.313;
   1:  PR[91,2] = PR[90,2] + 6.750;
   1:  PR[91,3] = PR[90,3] + 32.292;
   1:L PR[91] R[100]mm/sec CNT100;
   1:  PR[91,1] = PR[90,1] + 29.953;
   1:  PR[91,2] = PR[90,2] + 7.598;
   1:  PR[91,3] = PR[90,3] + 32.299;
   1:L PR[91] R[100]mm/sec CNT100;
   1:  PR[91,1] = PR[90,1] + 29.545;
   1:  PR[91,2] = PR[90,2] + 8.440;
   1:  PR[91,3] = PR[90,3] + 32.306;
   1:L PR[91] R[100]mm/sec CNT100;
   1:  PR[91,1] = PR[90,1] + 29.092;
   1:  PR[91,2] = PR[90,2] + 9.268;
   1:  PR[91,3] = PR[90,3] + 32.313;
   1:L PR[91] R[100]mm/sec CNT100;
   1:  PR[91,1] = PR[90,1] + 28.596;
   1:  PR[91,2] = PR[90,2] + 10.080;
   1:  PR[91,3] = PR[90,3] + 32.321;
   1:L PR[91] R[100]mm/sec CNT100;
   1:  PR[91,1] = PR[90,1] + 28.056;
   1:  PR[91,2] = PR[90,2] + 10.870;
   1:  PR[91,3] = PR[90,3] + 32.328;
   1:L PR[91] R[100]mm/sec CNT100;
   1:  PR[91,1] = PR[90,1] + 27.475;
   1:  PR[91,2] = PR[90,2] + 11.634;
   1:  PR[91,3] = PR[90,3] + 32.336;
   1:L PR[91] R[100]mm/sec CNT100;
   1:  PR[91,1] = PR[90,1] + 26.853;
   1:  PR[91,2] = PR[90,2] + 12.369;
   1:  PR[91,3] = PR[90,3] + 32.343;
   1:L PR[91] R[100]mm/sec CNT100;
   1:  PR[91,1] = PR[90,1] + 26.192;
   1:  PR[91,2] = PR[90,2] + 13.073;
   1:  PR[91,3] = PR[90,3] + 32.351;
   1:L PR[91] R[100]mm/sec CNT100;
   1:  PR[91,1] = PR[90,1] + 25.491;
   1:  PR[91,2] = PR[90,2] + 13.745;
   1:  PR[91,3] = PR[90,3] + 32.358;
   1:L PR[91] R[100]mm/sec CNT100;
   1:  PR[91,1] = PR[90,1] + 25.275;
   1:  PR[91,2] = PR[90,2] + 13.934;
   1:  PR[91,3] = PR[90,3] + 32.366;
   1:L PR[91] R[100]mm/sec CNT100;
   1:  PR[91,1] = PR[90,1] + 24.756;
   1:  PR[91,2] = PR[90,2] + 14.381;
   1:  PR[91,3] = PR[90,3] + 32.368;
   1:L PR[91] R[100]mm/sec CNT100;
   1:  PR[91,1] = PR[90,1] + 23.984;
   1:  PR[91,2] = PR[90,2] + 14.983;
   1:  PR[91,3] = PR[90,3] + 32.374;
   1:L PR[91] R[100]mm/sec CNT100;
   1:  PR[91,1] = PR[90,1] + 23.180;
   1:  PR[91,2] = PR[90,2] + 15.548;
   1:  PR[91,3] = PR[90,3] + 32.381;
   1:L PR[91] R[100]mm/sec CNT100;
   1:  PR[91,1] = PR[90,1] + 22.344;
   1:  PR[91,2] = PR[90,2] + 16.075;
   1:  PR[91,3] = PR[90,3] + 32.389;
   1:L PR[91] R[100]mm/sec CNT100;
   1:  PR[91,1] = PR[90,1] + 21.473;
   1:  PR[91,2] = PR[90,2] + 16.565;
   1:  PR[91,3] = PR[90,3] + 32.397;
   1:L PR[91] R[100]mm/sec CNT100;
   1:  PR[91,1] = PR[90,1] + 20.580;
   1:  PR[91,2] = PR[90,2] + 17.013;
   1:  PR[91,3] = PR[90,3] + 32.404;
   1:L PR[91] R[100]mm/sec CNT100;
   1:  PR[91,1] = PR[90,1] + 19.656;
   1:  PR[91,2] = PR[90,2] + 17.421;
   1:  PR[91,3] = PR[90,3] + 32.412;
   1:L PR[91] R[100]mm/sec CNT100;
   1:  PR[91,1] = PR[90,1] + 18.709;
   1:  PR[91,2] = PR[90,2] + 17.785;
   1:  PR[91,3] = PR[90,3] + 32.420;
   1:L PR[91] R[100]mm/sec CNT100;
   1:  PR[91,1] = PR[90,1] + 17.740;
   1:  PR[91,2] = PR[90,2] + 18.103;
   1:  PR[91,3] = PR[90,3] + 32.428;
   1:L PR[91] R[100]mm/sec CNT100;
   1:  PR[91,1] = PR[90,1] + 16.754;
   1:  PR[91,2] = PR[90,2] + 18.374;
   1:  PR[91,3] = PR[90,3] + 32.436;
   1:L PR[91] R[100]mm/sec CNT100;
   1:  PR[91,1] = PR[90,1] + 15.751;
   1:  PR[91,2] = PR[90,2] + 18.596;
   1:  PR[91,3] = PR[90,3] + 32.444;
   1:L PR[91] R[100]mm/sec CNT100;
   1:  PR[91,1] = PR[90,1] + 14.732;
   1:  PR[91,2] = PR[90,2] + 18.769;
   1:  PR[91,3] = PR[90,3] + 32.452;
   1:L PR[91] R[100]mm/sec CNT100;
   1:  PR[91,1] = PR[90,1] + 14.260;
   1:  PR[91,2] = PR[90,2] + 18.829;
   1:  PR[91,3] = PR[90,3] + 32.460;
   1:L PR[91] R[100]mm/sec CNT100;
   1:  PR[91,1] = PR[90,1] + 13.711;
   1:  PR[91,2] = PR[90,2] + 18.889;
   1:  PR[91,3] = PR[90,3] + 32.464;
   1:L PR[91] R[100]mm/sec CNT100;
   1:  PR[91,1] = PR[90,1] + 12.675;
   1:  PR[91,2] = PR[90,2] + 18.959;
   1:  PR[91,3] = PR[90,3] + 32.468;
   1:L PR[91] R[100]mm/sec CNT100;
   1:  PR[91,1] = PR[90,1] + 11.636;
   1:  PR[91,2] = PR[90,2] + 18.977;
   1:  PR[91,3] = PR[90,3] + 32.476;
   1:L PR[91] R[100]mm/sec CNT100;
   1:  PR[91,1] = PR[90,1] + 10.596;
   1:  PR[91,2] = PR[90,2] + 18.942;
   1:  PR[91,3] = PR[90,3] + 32.484;
   1:L PR[91] R[100]mm/sec CNT100;
   1:  PR[91,1] = PR[90,1] + 9.558;
   1:  PR[91,2] = PR[90,2] + 18.854;
   1:  PR[91,3] = PR[90,3] + 32.492;
   1:L PR[91] R[100]mm/sec CNT100;
   1:  PR[91,1] = PR[90,1] + 8.524;
   1:  PR[91,2] = PR[90,2] + 18.714;
   1:  PR[91,3] = PR[90,3] + 32.501;
   1:L PR[91] R[100]mm/sec CNT100;
   1:  PR[91,1] = PR[90,1] + 7.486;
   1:  PR[91,2] = PR[90,2] + 18.517;
   1:  PR[91,3] = PR[90,3] + 32.509;
   1:L PR[91] R[100]mm/sec CNT100;
   1:  PR[91,1] = PR[90,1] + 6.521;
   1:  PR[91,2] = PR[90,2] + 18.285;
   1:  PR[91,3] = PR[90,3] + 32.517;
   1:L PR[91] R[100]mm/sec CNT100;
   1:  PR[91,1] = PR[90,1] + 5.566;
   1:  PR[91,2] = PR[90,2] + 18.006;
   1:  PR[91,3] = PR[90,3] + 32.525;
   1:L PR[91] R[100]mm/sec CNT100;
   1:  PR[91,1] = PR[90,1] + 4.630;
   1:  PR[91,2] = PR[90,2] + 17.681;
   1:  PR[91,3] = PR[90,3] + 32.533;
   1:L PR[91] R[100]mm/sec CNT100;
   1:  PR[91,1] = PR[90,1] + 3.485;
   1:  PR[91,2] = PR[90,2] + 17.210;
   1:  PR[91,3] = PR[90,3] + 32.540;
   1:L PR[91] R[100]mm/sec CNT100;
   1:  PR[91,1] = PR[90,1] + 2.541;
   1:  PR[91,2] = PR[90,2] + 16.758;
   1:  PR[91,3] = PR[90,3] + 32.550;
   1:L PR[91] R[100]mm/sec CNT100;
   1:  PR[91,1] = PR[90,1] + 1.935;
   1:  PR[91,2] = PR[90,2] + 16.437;
   1:  PR[91,3] = PR[90,3] + 32.558;
   1:L PR[91] R[100]mm/sec CNT100;
   1:  PR[91,1] = PR[90,1] + 1.180;
   1:  PR[91,2] = PR[90,2] + 16.002;
   1:  PR[91,3] = PR[90,3] + 32.564;
   1:L PR[91] R[100]mm/sec CNT100;
   1:  PR[91,1] = PR[90,1] + 0.721;
   1:  PR[91,2] = PR[90,2] + 15.822;
   1:  PR[91,3] = PR[90,3] + 32.570;
   1:L PR[91] R[100]mm/sec CNT100;
   1:  PR[91,1] = PR[90,1] + 0.407;
   1:  PR[91,2] = PR[90,2] + 15.756;
   1:  PR[91,3] = PR[90,3] + 32.574;
   1:L PR[91] R[100]mm/sec CNT100;
   1:  PR[91,1] = PR[90,1] + 0.233;
   1:  PR[91,2] = PR[90,2] + 15.722;
   1:  PR[91,3] = PR[90,3] + 32.577;
   1:L PR[91] R[100]mm/sec CNT100;
   1:  PR[91,1] = PR[90,1] + -0.256;
   1:  PR[91,2] = PR[90,2] + 15.702;
   1:  PR[91,3] = PR[90,3] + 32.578;
   1:L PR[91] R[100]mm/sec CNT100;
   1:  PR[91,1] = PR[90,1] + -0.744;
   1:  PR[91,2] = PR[90,2] + 15.765;
   1:  PR[91,3] = PR[90,3] + 32.582;
   1:L PR[91] R[100]mm/sec CNT100;
   1:  PR[91,1] = PR[90,1] + -1.215;
   1:  PR[91,2] = PR[90,2] + 15.909;
   1:  PR[91,3] = PR[90,3] + 32.586;
   1:L PR[91] R[100]mm/sec CNT100;
   1:  PR[91,1] = PR[90,1] + -1.630;
   1:  PR[91,2] = PR[90,2] + 16.116;
   1:  PR[91,3] = PR[90,3] + 32.590;
   1:L PR[91] R[100]mm/sec CNT100;
   1:  PR[91,1] = PR[90,1] + -2.177;
   1:  PR[91,2] = PR[90,2] + 16.436;
   1:  PR[91,3] = PR[90,3] + 32.593;
   1:L PR[91] R[100]mm/sec CNT100;
   1:  PR[91,1] = PR[90,1] + -3.053;
   1:  PR[91,2] = PR[90,2] + 16.896;
   1:  PR[91,3] = PR[90,3] + 32.598;
   1:L PR[91] R[100]mm/sec CNT100;
   1:  PR[91,1] = PR[90,1] + -3.952;
   1:  PR[91,2] = PR[90,2] + 17.312;
   1:  PR[91,3] = PR[90,3] + 32.606;
   1:L PR[91] R[100]mm/sec CNT100;
   1:  PR[91,1] = PR[90,1] + -4.871;
   1:  PR[91,2] = PR[90,2] + 17.683;
   1:  PR[91,3] = PR[90,3] + 32.614;
   1:L PR[91] R[100]mm/sec CNT100;
   1:  PR[91,1] = PR[90,1] + -5.809;
   1:  PR[91,2] = PR[90,2] + 18.009;
   1:  PR[91,3] = PR[90,3] + 32.621;
   1:L PR[91] R[100]mm/sec CNT100;
   1:  PR[91,1] = PR[90,1] + -6.763;
   1:  PR[91,2] = PR[90,2] + 18.288;
   1:  PR[91,3] = PR[90,3] + 32.629;
   1:L PR[91] R[100]mm/sec CNT100;
   1:  PR[91,1] = PR[90,1] + -7.740;
   1:  PR[91,2] = PR[90,2] + 18.522;
   1:  PR[91,3] = PR[90,3] + 32.637;
   1:L PR[91] R[100]mm/sec CNT100;
   1:  PR[91,1] = PR[90,1] + -8.767;
   1:  PR[91,2] = PR[90,2] + 18.715;
   1:  PR[91,3] = PR[90,3] + 32.645;
   1:L PR[91] R[100]mm/sec CNT100;
   1:  PR[91,1] = PR[90,1] + -9.800;
   1:  PR[91,2] = PR[90,2] + 18.855;
   1:  PR[91,3] = PR[90,3] + 32.653;
   1:L PR[91] R[100]mm/sec CNT100;
   1:  PR[91,1] = PR[90,1] + -10.840;
   1:  PR[91,2] = PR[90,2] + 18.942;
   1:  PR[91,3] = PR[90,3] + 32.661;
   1:L PR[91] R[100]mm/sec CNT100;
   1:  PR[91,1] = PR[90,1] + -11.600;
   1:  PR[91,2] = PR[90,2] + 18.971;
   1:  PR[91,3] = PR[90,3] + 32.669;
   1:L PR[91] R[100]mm/sec CNT100;
   1:  PR[91,1] = PR[90,1] + -12.573;
   1:  PR[91,2] = PR[90,2] + 18.969;
   1:  PR[91,3] = PR[90,3] + 32.675;
   1:L PR[91] R[100]mm/sec CNT100;
   1:  PR[91,1] = PR[90,1] + -13.539;
   1:  PR[91,2] = PR[90,2] + 18.921;
   1:  PR[91,3] = PR[90,3] + 32.683;
   1:L PR[91] R[100]mm/sec CNT100;
   1:  PR[91,1] = PR[90,1] + -14.500;
   1:  PR[91,2] = PR[90,2] + 18.828;
   1:  PR[91,3] = PR[90,3] + 32.690;
   1:L PR[91] R[100]mm/sec CNT100;
   1:  PR[91,1] = PR[90,1] + -15.456;
   1:  PR[91,2] = PR[90,2] + 18.690;
   1:  PR[91,3] = PR[90,3] + 32.698;
   1:L PR[91] R[100]mm/sec CNT100;
   1:  PR[91,1] = PR[90,1] + -15.990;
   1:  PR[91,2] = PR[90,2] + 18.596;
   1:  PR[91,3] = PR[90,3] + 32.705;
   1:L PR[91] R[100]mm/sec CNT100;
   1:  PR[91,1] = PR[90,1] + -16.995;
   1:  PR[91,2] = PR[90,2] + 18.374;
   1:  PR[91,3] = PR[90,3] + 32.710;
   1:L PR[91] R[100]mm/sec CNT100;
   1:  PR[91,1] = PR[90,1] + -17.982;
   1:  PR[91,2] = PR[90,2] + 18.104;
   1:  PR[91,3] = PR[90,3] + 32.718;
   1:L PR[91] R[100]mm/sec CNT100;
   1:  PR[91,1] = PR[90,1] + -18.949;
   1:  PR[91,2] = PR[90,2] + 17.786;
   1:  PR[91,3] = PR[90,3] + 32.726;
   1:L PR[91] R[100]mm/sec CNT100;
   1:  PR[91,1] = PR[90,1] + -19.896;
   1:  PR[91,2] = PR[90,2] + 17.422;
   1:  PR[91,3] = PR[90,3] + 32.734;
   1:L PR[91] R[100]mm/sec CNT100;
   1:  PR[91,1] = PR[90,1] + -20.819;
   1:  PR[91,2] = PR[90,2] + 17.013;
   1:  PR[91,3] = PR[90,3] + 32.742;
   1:L PR[91] R[100]mm/sec CNT100;
   1:  PR[91,1] = PR[90,1] + -21.720;
   1:  PR[91,2] = PR[90,2] + 16.559;
   1:  PR[91,3] = PR[90,3] + 32.750;
   1:L PR[91] R[100]mm/sec CNT100;
   1:  PR[91,1] = PR[90,1] + -22.556;
   1:  PR[91,2] = PR[90,2] + 16.088;
   1:  PR[91,3] = PR[90,3] + 32.757;
   1:L PR[91] R[100]mm/sec CNT100;
   1:  PR[91,1] = PR[90,1] + -23.373;
   1:  PR[91,2] = PR[90,2] + 15.575;
   1:  PR[91,3] = PR[90,3] + 32.765;
   1:L PR[91] R[100]mm/sec CNT100;
   1:  PR[91,1] = PR[90,1] + -24.162;
   1:  PR[91,2] = PR[90,2] + 15.024;
   1:  PR[91,3] = PR[90,3] + 32.772;
   1:L PR[91] R[100]mm/sec CNT100;
   1:  PR[91,1] = PR[90,1] + -24.922;
   1:  PR[91,2] = PR[90,2] + 14.437;
   1:  PR[91,3] = PR[90,3] + 32.780;
   1:L PR[91] R[100]mm/sec CNT100;
   1:  PR[91,1] = PR[90,1] + -25.651;
   1:  PR[91,2] = PR[90,2] + 13.814;
   1:  PR[91,3] = PR[90,3] + 32.787;
   1:L PR[91] R[100]mm/sec CNT100;
   1:  PR[91,1] = PR[90,1] + -26.348;
   1:  PR[91,2] = PR[90,2] + 13.155;
   1:  PR[91,3] = PR[90,3] + 32.795;
   1:L PR[91] R[100]mm/sec CNT100;
   1:  PR[91,1] = PR[90,1] + -26.610;
   1:  PR[91,2] = PR[90,2] + 12.886;
   1:  PR[91,3] = PR[90,3] + 32.802;
   1:L PR[91] R[100]mm/sec CNT100;
   1:  PR[91,1] = PR[90,1] + -27.007;
   1:  PR[91,2] = PR[90,2] + 12.467;
   1:  PR[91,3] = PR[90,3] + 32.805;
   1:L PR[91] R[100]mm/sec CNT100;
   1:  PR[91,1] = PR[90,1] + -27.632;
   1:  PR[91,2] = PR[90,2] + 11.742;
   1:  PR[91,3] = PR[90,3] + 32.810;
   1:L PR[91] R[100]mm/sec CNT100;
   1:  PR[91,1] = PR[90,1] + -28.217;
   1:  PR[91,2] = PR[90,2] + 10.987;
   1:  PR[91,3] = PR[90,3] + 32.817;
   1:L PR[91] R[100]mm/sec CNT100;
   1:  PR[91,1] = PR[90,1] + -28.762;
   1:  PR[91,2] = PR[90,2] + 10.201;
   1:  PR[91,3] = PR[90,3] + 32.825;
   1:L PR[91] R[100]mm/sec CNT100;
   1:  PR[91,1] = PR[90,1] + -29.265;
   1:  PR[91,2] = PR[90,2] + 9.389;
   1:  PR[91,3] = PR[90,3] + 32.832;
   1:L PR[91] R[100]mm/sec CNT100;
   1:  PR[91,1] = PR[90,1] + -29.726;
   1:  PR[91,2] = PR[90,2] + 8.554;
   1:  PR[91,3] = PR[90,3] + 32.840;
   1:L PR[91] R[100]mm/sec CNT100;
   1:  PR[91,1] = PR[90,1] + -30.143;
   1:  PR[91,2] = PR[90,2] + 7.701;
   1:  PR[91,3] = PR[90,3] + 32.847;
   1:L PR[91] R[100]mm/sec CNT100;
   1:  PR[91,1] = PR[90,1] + -30.408;
   1:  PR[91,2] = PR[90,2] + 7.085;
   1:  PR[91,3] = PR[90,3] + 32.855;
   1:L PR[91] R[100]mm/sec CNT100;
   1:  PR[91,1] = PR[90,1] + -30.837;
   1:  PR[91,2] = PR[90,2] + 5.964;
   1:  PR[91,3] = PR[90,3] + 32.860;
   1:L PR[91] R[100]mm/sec CNT100;
   1:  PR[91,1] = PR[90,1] + -31.110;
   1:  PR[91,2] = PR[90,2] + 5.089;
   1:  PR[91,3] = PR[90,3] + 32.869;
   1:L PR[91] R[100]mm/sec CNT100;
   1:  PR[91,1] = PR[90,1] + -31.336;
   1:  PR[91,2] = PR[90,2] + 4.204;
   1:  PR[91,3] = PR[90,3] + 32.876;
   1:L PR[91] R[100]mm/sec CNT100;
   1:  PR[91,1] = PR[90,1] + -31.511;
   1:  PR[91,2] = PR[90,2] + 3.303;
   1:  PR[91,3] = PR[90,3] + 32.884;
   1:L PR[91] R[100]mm/sec CNT100;
   1:  PR[91,1] = PR[90,1] + -31.638;
   1:  PR[91,2] = PR[90,2] + 2.379;
   1:  PR[91,3] = PR[90,3] + 32.891;
   1:L PR[91] R[100]mm/sec CNT100;
   1:  PR[91,1] = PR[90,1] + -31.714;
   1:  PR[91,2] = PR[90,2] + 1.423;
   1:  PR[91,3] = PR[90,3] + 32.898;
   1:L PR[91] R[100]mm/sec CNT100;
   1:  PR[91,1] = PR[90,1] + -31.739;
   1:  PR[91,2] = PR[90,2] + 0.428;
   1:  PR[91,3] = PR[90,3] + 32.906;
   1:L PR[91] R[100]mm/sec CNT100;
   1:  PR[91,1] = PR[90,1] + -31.714;
   1:  PR[91,2] = PR[90,2] + -0.568;
   1:  PR[91,3] = PR[90,3] + 32.913;
   1:L PR[91] R[100]mm/sec CNT100;
   1:  PR[91,1] = PR[90,1] + -31.638;
   1:  PR[91,2] = PR[90,2] + -1.524;
   1:  PR[91,3] = PR[90,3] + 32.921;
   1:L PR[91] R[100]mm/sec CNT100;
   1:  PR[91,1] = PR[90,1] + -31.511;
   1:  PR[91,2] = PR[90,2] + -2.448;
   1:  PR[91,3] = PR[90,3] + 32.929;
   1:L PR[91] R[100]mm/sec CNT100;
   1:  PR[91,1] = PR[90,1] + -31.336;
   1:  PR[91,2] = PR[90,2] + -3.348;
   1:  PR[91,3] = PR[90,3] + 32.936;
   1:L PR[91] R[100]mm/sec CNT100;
   1:  PR[91,1] = PR[90,1] + -31.110;
   1:  PR[91,2] = PR[90,2] + -4.234;
   1:  PR[91,3] = PR[90,3] + 32.943;
   1:L PR[91] R[100]mm/sec CNT100;
   1:  PR[91,1] = PR[90,1] + -30.836;
   1:  PR[91,2] = PR[90,2] + -5.112;
   1:  PR[91,3] = PR[90,3] + 32.950;
   1:L PR[91] R[100]mm/sec CNT100;
   1:  PR[91,1] = PR[90,1] + -30.513;
   1:  PR[91,2] = PR[90,2] + -5.982;
   1:  PR[91,3] = PR[90,3] + 32.957;
   1:L PR[91] R[100]mm/sec CNT100;
   1:  PR[91,1] = PR[90,1] + -30.142;
   1:  PR[91,2] = PR[90,2] + -6.847;
   1:  PR[91,3] = PR[90,3] + 32.965;
   1:L PR[91] R[100]mm/sec CNT100;
   1:  PR[91,1] = PR[90,1] + -30.014;
   1:  PR[91,2] = PR[90,2] + -7.112;
   1:  PR[91,3] = PR[90,3] + 32.972;
   1:L PR[91] R[100]mm/sec CNT100;
   1:  PR[91,1] = PR[90,1] + -29.726;
   1:  PR[91,2] = PR[90,2] + -7.698;
   1:  PR[91,3] = PR[90,3] + 32.974;
   1:L PR[91] R[100]mm/sec CNT100;
   1:  PR[91,1] = PR[90,1] + -29.265;
   1:  PR[91,2] = PR[90,2] + -8.533;
   1:  PR[91,3] = PR[90,3] + 32.979;
   1:L PR[91] R[100]mm/sec CNT100;
   1:  PR[91,1] = PR[90,1] + -28.762;
   1:  PR[91,2] = PR[90,2] + -9.346;
   1:  PR[91,3] = PR[90,3] + 32.987;
   1:L PR[91] R[100]mm/sec CNT100;
   1:  PR[91,1] = PR[90,1] + -28.217;
   1:  PR[91,2] = PR[90,2] + -10.132;
   1:  PR[91,3] = PR[90,3] + 32.994;
   1:L PR[91] R[100]mm/sec CNT100;
   1:  PR[91,1] = PR[90,1] + -27.631;
   1:  PR[91,2] = PR[90,2] + -10.888;
   1:  PR[91,3] = PR[90,3] + 33.002;
   1:L PR[91] R[100]mm/sec CNT100;
   1:  PR[91,1] = PR[90,1] + -27.292;
   1:  PR[91,2] = PR[90,2] + -11.285;
   1:  PR[91,3] = PR[90,3] + 33.009;
   1:L PR[91] R[100]mm/sec CNT100;
   1:  PR[91,1] = PR[90,1] + -27.009;
   1:  PR[91,2] = PR[90,2] + -11.609;
   1:  PR[91,3] = PR[90,3] + 33.013;
   1:L PR[91] R[100]mm/sec CNT100;
   1:  PR[91,1] = PR[90,1] + -26.347;
   1:  PR[91,2] = PR[90,2] + -12.302;
   1:  PR[91,3] = PR[90,3] + 33.017;
   1:L PR[91] R[100]mm/sec CNT100;
   1:  PR[91,1] = PR[90,1] + -25.651;
   1:  PR[91,2] = PR[90,2] + -12.959;
   1:  PR[91,3] = PR[90,3] + 33.024;
   1:L PR[91] R[100]mm/sec CNT100;
   1:  PR[91,1] = PR[90,1] + -24.923;
   1:  PR[91,2] = PR[90,2] + -13.582;
   1:  PR[91,3] = PR[90,3] + 33.032;
   1:L PR[91] R[100]mm/sec CNT100;
   1:  PR[91,1] = PR[90,1] + -24.163;
   1:  PR[91,2] = PR[90,2] + -14.169;
   1:  PR[91,3] = PR[90,3] + 33.039;
   1:L PR[91] R[100]mm/sec CNT100;
   1:  PR[91,1] = PR[90,1] + -23.373;
   1:  PR[91,2] = PR[90,2] + -14.720;
   1:  PR[91,3] = PR[90,3] + 33.047;
   1:L PR[91] R[100]mm/sec CNT100;
   1:  PR[91,1] = PR[90,1] + -22.557;
   1:  PR[91,2] = PR[90,2] + -15.232;
   1:  PR[91,3] = PR[90,3] + 33.054;
   1:L PR[91] R[100]mm/sec CNT100;
   1:  PR[91,1] = PR[90,1] + -21.716;
   1:  PR[91,2] = PR[90,2] + -15.706;
   1:  PR[91,3] = PR[90,3] + 33.062;
   1:L PR[91] R[100]mm/sec CNT100;
   1:  PR[91,1] = PR[90,1] + -20.820;
   1:  PR[91,2] = PR[90,2] + -16.157;
   1:  PR[91,3] = PR[90,3] + 33.069;
   1:L PR[91] R[100]mm/sec CNT100;
   1:  PR[91,1] = PR[90,1] + -19.897;
   1:  PR[91,2] = PR[90,2] + -16.566;
   1:  PR[91,3] = PR[90,3] + 33.077;
   1:L PR[91] R[100]mm/sec CNT100;
   1:  PR[91,1] = PR[90,1] + -18.950;
   1:  PR[91,2] = PR[90,2] + -16.931;
   1:  PR[91,3] = PR[90,3] + 33.085;
   1:L PR[91] R[100]mm/sec CNT100;
   1:  PR[91,1] = PR[90,1] + -17.982;
   1:  PR[91,2] = PR[90,2] + -17.249;
   1:  PR[91,3] = PR[90,3] + 33.093;
   1:L PR[91] R[100]mm/sec CNT100;
   1:  PR[91,1] = PR[90,1] + -16.994;
   1:  PR[91,2] = PR[90,2] + -17.519;
   1:  PR[91,3] = PR[90,3] + 33.101;
   1:L PR[91] R[100]mm/sec CNT100;
   1:  PR[91,1] = PR[90,1] + -16.398;
   1:  PR[91,2] = PR[90,2] + -17.655;
   1:  PR[91,3] = PR[90,3] + 33.109;
   1:L PR[91] R[100]mm/sec CNT100;
   1:  PR[91,1] = PR[90,1] + -15.452;
   1:  PR[91,2] = PR[90,2] + -17.836;
   1:  PR[91,3] = PR[90,3] + 33.114;
   1:L PR[91] R[100]mm/sec CNT100;
   1:  PR[91,1] = PR[90,1] + -14.500;
   1:  PR[91,2] = PR[90,2] + -17.973;
   1:  PR[91,3] = PR[90,3] + 33.121;
   1:L PR[91] R[100]mm/sec CNT100;
   1:  PR[91,1] = PR[90,1] + -13.540;
   1:  PR[91,2] = PR[90,2] + -18.066;
   1:  PR[91,3] = PR[90,3] + 33.129;
   1:L PR[91] R[100]mm/sec CNT100;
   1:  PR[91,1] = PR[90,1] + -12.573;
   1:  PR[91,2] = PR[90,2] + -18.113;
   1:  PR[91,3] = PR[90,3] + 33.136;
   1:L PR[91] R[100]mm/sec CNT100;
   1:  PR[91,1] = PR[90,1] + -11.602;
   1:  PR[91,2] = PR[90,2] + -18.116;
   1:  PR[91,3] = PR[90,3] + 33.144;
   1:L PR[91] R[100]mm/sec CNT100;
   1:  PR[91,1] = PR[90,1] + -10.629;
   1:  PR[91,2] = PR[90,2] + -18.072;
   1:  PR[91,3] = PR[90,3] + 33.151;
   1:L PR[91] R[100]mm/sec CNT100;
   1:  PR[91,1] = PR[90,1] + -9.802;
   1:  PR[91,2] = PR[90,2] + -18.000;
   1:  PR[91,3] = PR[90,3] + 33.159;
   1:L PR[91] R[100]mm/sec CNT100;
   1:  PR[91,1] = PR[90,1] + -8.690;
   1:  PR[91,2] = PR[90,2] + -17.847;
   1:  PR[91,3] = PR[90,3] + 33.166;
   1:L PR[91] R[100]mm/sec CNT100;
   1:  PR[91,1] = PR[90,1] + -7.729;
   1:  PR[91,2] = PR[90,2] + -17.664;
   1:  PR[91,3] = PR[90,3] + 33.174;
   1:L PR[91] R[100]mm/sec CNT100;
   1:  PR[91,1] = PR[90,1] + -6.763;
   1:  PR[91,2] = PR[90,2] + -17.433;
   1:  PR[91,3] = PR[90,3] + 33.182;
   1:L PR[91] R[100]mm/sec CNT100;
   1:  PR[91,1] = PR[90,1] + -5.809;
   1:  PR[91,2] = PR[90,2] + -17.154;
   1:  PR[91,3] = PR[90,3] + 33.190;
   1:L PR[91] R[100]mm/sec CNT100;
   1:  PR[91,1] = PR[90,1] + -4.871;
   1:  PR[91,2] = PR[90,2] + -16.828;
   1:  PR[91,3] = PR[90,3] + 33.198;
   1:L PR[91] R[100]mm/sec CNT100;
   1:  PR[91,1] = PR[90,1] + -3.952;
   1:  PR[91,2] = PR[90,2] + -16.457;
   1:  PR[91,3] = PR[90,3] + 33.205;
   1:L PR[91] R[100]mm/sec CNT100;
   1:  PR[91,1] = PR[90,1] + -3.054;
   1:  PR[91,2] = PR[90,2] + -16.041;
   1:  PR[91,3] = PR[90,3] + 33.213;
   1:L PR[91] R[100]mm/sec CNT100;
   1:  PR[91,1] = PR[90,1] + -2.178;
   1:  PR[91,2] = PR[90,2] + -15.581;
   1:  PR[91,3] = PR[90,3] + 33.221;
   1:L PR[91] R[100]mm/sec CNT100;
   1:  PR[91,1] = PR[90,1] + -1.630;
   1:  PR[91,2] = PR[90,2] + -15.261;
   1:  PR[91,3] = PR[90,3] + 33.229;
   1:L PR[91] R[100]mm/sec CNT100;
   1:  PR[91,1] = PR[90,1] + -1.214;
   1:  PR[91,2] = PR[90,2] + -15.053;
   1:  PR[91,3] = PR[90,3] + 33.233;
   1:L PR[91] R[100]mm/sec CNT100;
   1:  PR[91,1] = PR[90,1] + -0.744;
   1:  PR[91,2] = PR[90,2] + -14.910;
   1:  PR[91,3] = PR[90,3] + 33.237;
   1:L PR[91] R[100]mm/sec CNT100;
   1:  PR[91,1] = PR[90,1] + -0.256;
   1:  PR[91,2] = PR[90,2] + -14.847;
   1:  PR[91,3] = PR[90,3] + 33.241;
   1:L PR[91] R[100]mm/sec CNT100;
   1:  PR[91,1] = PR[90,1] + 0.233;
   1:  PR[91,2] = PR[90,2] + -14.867;
   1:  PR[91,3] = PR[90,3] + 33.245;
   1:L PR[91] R[100]mm/sec CNT100;
   1:  PR[91,1] = PR[90,1] + 0.407;
   1:  PR[91,2] = PR[90,2] + -14.901;
   1:  PR[91,3] = PR[90,3] + 33.249;
   1:L PR[91] R[100]mm/sec CNT100;
   1:  PR[91] = PR[90];
   1:  PR[91,1] = PR[90,1] + 0.803;
   1:  PR[91,2] = PR[90,2] + -15.481;
   1:  PR[91,3] = PR[90,3] + 34.580;
   1:L PR[91] R[100]mm/sec CNT100;
   1:  PR[91,1] = PR[90,1] + 1.245;
   1:  PR[91,2] = PR[90,2] + -15.667;
   1:  PR[91,3] = PR[90,3] + 33.254;
   1:L PR[91] R[100]mm/sec CNT100;
   1:  PR[91,1] = PR[90,1] + 1.702;
   1:  PR[91,2] = PR[90,2] + -15.919;
   1:  PR[91,3] = PR[90,3] + 33.258;
   1:L PR[91] R[100]mm/sec CNT100;
   1:  PR[91,1] = PR[90,1] + 2.386;
   1:  PR[91,2] = PR[90,2] + -16.267;
   1:  PR[91,3] = PR[90,3] + 33.262;
   1:L PR[91] R[100]mm/sec CNT100;
   1:  PR[91,1] = PR[90,1] + 3.292;
   1:  PR[91,2] = PR[90,2] + -16.676;
   1:  PR[91,3] = PR[90,3] + 33.268;
   1:L PR[91] R[100]mm/sec CNT100;
   1:  PR[91,1] = PR[90,1] + 4.218;
   1:  PR[91,2] = PR[90,2] + -17.041;
   1:  PR[91,3] = PR[90,3] + 33.276;
   1:L PR[91] R[100]mm/sec CNT100;
   1:  PR[91,1] = PR[90,1] + 5.162;
   1:  PR[91,2] = PR[90,2] + -17.361;
   1:  PR[91,3] = PR[90,3] + 33.284;
   1:L PR[91] R[100]mm/sec CNT100;
   1:  PR[91,1] = PR[90,1] + 6.124;
   1:  PR[91,2] = PR[90,2] + -17.634;
   1:  PR[91,3] = PR[90,3] + 33.291;
   1:L PR[91] R[100]mm/sec CNT100;
   1:  PR[91,1] = PR[90,1] + 6.633;
   1:  PR[91,2] = PR[90,2] + -17.757;
   1:  PR[91,3] = PR[90,3] + 33.299;
   1:L PR[91] R[100]mm/sec CNT100;
   1:  PR[91,1] = PR[90,1] + 7.092;
   1:  PR[91,2] = PR[90,2] + -17.859;
   1:  PR[91,3] = PR[90,3] + 33.303;
   1:L PR[91] R[100]mm/sec CNT100;
   1:  PR[91,1] = PR[90,1] + 8.079;
   1:  PR[91,2] = PR[90,2] + -18.038;
   1:  PR[91,3] = PR[90,3] + 33.307;
   1:L PR[91] R[100]mm/sec CNT100;
   1:  PR[91,1] = PR[90,1] + 9.071;
   1:  PR[91,2] = PR[90,2] + -18.168;
   1:  PR[91,3] = PR[90,3] + 33.315;
   1:L PR[91] R[100]mm/sec CNT100;
   1:  PR[91,1] = PR[90,1] + 10.069;
   1:  PR[91,2] = PR[90,2] + -18.250;
   1:  PR[91,3] = PR[90,3] + 33.323;
   1:L PR[91] R[100]mm/sec CNT100;
   1:  PR[91,1] = PR[90,1] + 11.071;
   1:  PR[91,2] = PR[90,2] + -18.283;
   1:  PR[91,3] = PR[90,3] + 33.331;
   1:L PR[91] R[100]mm/sec CNT100;
   1:  PR[91,1] = PR[90,1] + 11.938;
   1:  PR[91,2] = PR[90,2] + -18.270;
   1:  PR[91,3] = PR[90,3] + 33.339;
   1:L PR[91] R[100]mm/sec CNT100;
   1:  PR[91,1] = PR[90,1] + 13.075;
   1:  PR[91,2] = PR[90,2] + -18.202;
   1:  PR[91,3] = PR[90,3] + 33.346;
   1:L PR[91] R[100]mm/sec CNT100;
   1:  PR[91,1] = PR[90,1] + 14.077;
   1:  PR[91,2] = PR[90,2] + -18.089;
   1:  PR[91,3] = PR[90,3] + 33.355;
   1:L PR[91] R[100]mm/sec CNT100;
   1:  PR[91,1] = PR[90,1] + 15.106;
   1:  PR[91,2] = PR[90,2] + -17.923;
   1:  PR[91,3] = PR[90,3] + 33.363;
   1:L PR[91] R[100]mm/sec CNT100;
   1:  PR[91,1] = PR[90,1] + 16.122;
   1:  PR[91,2] = PR[90,2] + -17.705;
   1:  PR[91,3] = PR[90,3] + 33.371;
   1:L PR[91] R[100]mm/sec CNT100;
   1:  PR[91,1] = PR[90,1] + 17.122;
   1:  PR[91,2] = PR[90,2] + -17.438;
   1:  PR[91,3] = PR[90,3] + 33.379;
   1:L PR[91] R[100]mm/sec CNT100;
   1:  PR[91,1] = PR[90,1] + 18.103;
   1:  PR[91,2] = PR[90,2] + -17.122;
   1:  PR[91,3] = PR[90,3] + 33.387;
   1:L PR[91] R[100]mm/sec CNT100;
   1:  PR[91,1] = PR[90,1] + 19.064;
   1:  PR[91,2] = PR[90,2] + -16.760;
   1:  PR[91,3] = PR[90,3] + 33.395;
   1:L PR[91] R[100]mm/sec CNT100;
   1:  PR[91,1] = PR[90,1] + 20.001;
   1:  PR[91,2] = PR[90,2] + -16.352;
   1:  PR[91,3] = PR[90,3] + 33.403;
   1:L PR[91] R[100]mm/sec CNT100;
   1:  PR[91,1] = PR[90,1] + 20.912;
   1:  PR[91,2] = PR[90,2] + -15.901;
   1:  PR[91,3] = PR[90,3] + 33.411;
   1:L PR[91] R[100]mm/sec CNT100;
   1:  PR[91,1] = PR[90,1] + 21.796;
   1:  PR[91,2] = PR[90,2] + -15.406;
   1:  PR[91,3] = PR[90,3] + 33.419;
   1:L PR[91] R[100]mm/sec CNT100;
   1:  PR[91,1] = PR[90,1] + 22.151;
   1:  PR[91,2] = PR[90,2] + -15.187;
   1:  PR[91,3] = PR[90,3] + 33.427;
   1:L PR[91] R[100]mm/sec CNT100;
   1:  PR[91,1] = PR[90,1] + 22.646;
   1:  PR[91,2] = PR[90,2] + -14.874;
   1:  PR[91,3] = PR[90,3] + 33.431;
   1:L PR[91] R[100]mm/sec CNT100;
   1:  PR[91,1] = PR[90,1] + 23.466;
   1:  PR[91,2] = PR[90,2] + -14.300;
   1:  PR[91,3] = PR[90,3] + 33.435;
   1:L PR[91] R[100]mm/sec CNT100;
   1:  PR[91,1] = PR[90,1] + 24.251;
   1:  PR[91,2] = PR[90,2] + -13.690;
   1:  PR[91,3] = PR[90,3] + 33.443;
   1:L PR[91] R[100]mm/sec CNT100;
   1:  PR[91,1] = PR[90,1] + 25.000;
   1:  PR[91,2] = PR[90,2] + -13.044;
   1:  PR[91,3] = PR[90,3] + 33.451;
   1:L PR[91] R[100]mm/sec CNT100;
   1:  PR[91,1] = PR[90,1] + 25.711;
   1:  PR[91,2] = PR[90,2] + -12.364;
   1:  PR[91,3] = PR[90,3] + 33.459;
   1:L PR[91] R[100]mm/sec CNT100;
   1:  PR[91,1] = PR[90,1] + 26.383;
   1:  PR[91,2] = PR[90,2] + -11.650;
   1:  PR[91,3] = PR[90,3] + 33.467;
   1:L PR[91] R[100]mm/sec CNT100;
   1:  PR[91,1] = PR[90,1] + 27.014;
   1:  PR[91,2] = PR[90,2] + -10.905;
   1:  PR[91,3] = PR[90,3] + 33.474;
   1:L PR[91] R[100]mm/sec CNT100;
   1:  PR[91,1] = PR[90,1] + 27.603;
   1:  PR[91,2] = PR[90,2] + -10.131;
   1:  PR[91,3] = PR[90,3] + 33.482;
   1:L PR[91] R[100]mm/sec CNT100;
   1:  PR[91,1] = PR[90,1] + 28.150;
   1:  PR[91,2] = PR[90,2] + -9.334;
   1:  PR[91,3] = PR[90,3] + 33.490;
   1:L PR[91] R[100]mm/sec CNT100;
   1:  PR[91,1] = PR[90,1] + 28.653;
   1:  PR[91,2] = PR[90,2] + -8.514;
   1:  PR[91,3] = PR[90,3] + 33.497;
   1:L PR[91] R[100]mm/sec CNT100;
   1:  PR[91,1] = PR[90,1] + 29.111;
   1:  PR[91,2] = PR[90,2] + -7.676;
   1:  PR[91,3] = PR[90,3] + 33.505;
   1:L PR[91] R[100]mm/sec CNT100;
   1:  PR[91,1] = PR[90,1] + 29.524;
   1:  PR[91,2] = PR[90,2] + -6.826;
   1:  PR[91,3] = PR[90,3] + 33.513;
   1:L PR[91] R[100]mm/sec CNT100;
   1:  PR[91,1] = PR[90,1] + 29.890;
   1:  PR[91,2] = PR[90,2] + -5.967;
   1:  PR[91,3] = PR[90,3] + 33.520;
   1:L PR[91] R[100]mm/sec CNT100;
   1:  PR[91,1] = PR[90,1] + 30.208;
   1:  PR[91,2] = PR[90,2] + -5.102;
   1:  PR[91,3] = PR[90,3] + 33.527;
   1:L PR[91] R[100]mm/sec CNT100;
   1:  PR[91,1] = PR[90,1] + 30.477;
   1:  PR[91,2] = PR[90,2] + -4.229;
   1:  PR[91,3] = PR[90,3] + 33.535;
   1:L PR[91] R[100]mm/sec CNT100;
   1:  PR[91,1] = PR[90,1] + 30.698;
   1:  PR[91,2] = PR[90,2] + -3.343;
   1:  PR[91,3] = PR[90,3] + 33.542;
   1:L PR[91] R[100]mm/sec CNT100;
   1:  PR[91,1] = PR[90,1] + 30.871;
   1:  PR[91,2] = PR[90,2] + -2.441;
   1:  PR[91,3] = PR[90,3] + 33.549;
   1:L PR[91] R[100]mm/sec CNT100;
   1:  PR[91,1] = PR[90,1] + 30.995;
   1:  PR[91,2] = PR[90,2] + -1.515;
   1:  PR[91,3] = PR[90,3] + 33.556;
   1:L PR[91] R[100]mm/sec CNT100;
   1:  PR[91,1] = PR[90,1] + 31.069;
   1:  PR[91,2] = PR[90,2] + -0.561;
   1:  PR[91,3] = PR[90,3] + 33.564;
   1:L PR[91] R[100]mm/sec CNT100;
   1:  PR[91,1] = PR[90,1] + 31.094;
   1:  PR[91,2] = PR[90,2] + 0.428;
   1:  PR[91,3] = PR[90,3] + 33.571;
   1:L PR[91] R[100]mm/sec CNT100;
   1:  PR[91,1] = PR[90,1] + 31.069;
   1:  PR[91,2] = PR[90,2] + 1.416;
   1:  PR[91,3] = PR[90,3] + 33.579;
   1:L PR[91] R[100]mm/sec CNT100;
   1:  PR[91,1] = PR[90,1] + 30.995;
   1:  PR[91,2] = PR[90,2] + 2.370;
   1:  PR[91,3] = PR[90,3] + 33.587;
   1:L PR[91] R[100]mm/sec CNT100;
   1:  PR[91,1] = PR[90,1] + 30.871;
   1:  PR[91,2] = PR[90,2] + 3.296;
   1:  PR[91,3] = PR[90,3] + 33.594;
   1:L PR[91] R[100]mm/sec CNT100;
   1:  PR[91,1] = PR[90,1] + 30.698;
   1:  PR[91,2] = PR[90,2] + 4.199;
   1:  PR[91,3] = PR[90,3] + 33.602;
   1:L PR[91] R[100]mm/sec CNT100;
   1:  PR[91,1] = PR[90,1] + 30.477;
   1:  PR[91,2] = PR[90,2] + 5.084;
   1:  PR[91,3] = PR[90,3] + 33.609;
   1:L PR[91] R[100]mm/sec CNT100;
   1:  PR[91,1] = PR[90,1] + 30.208;
   1:  PR[91,2] = PR[90,2] + 5.958;
   1:  PR[91,3] = PR[90,3] + 33.616;
   1:L PR[91] R[100]mm/sec CNT100;
   1:  PR[91,1] = PR[90,1] + 29.890;
   1:  PR[91,2] = PR[90,2] + 6.823;
   1:  PR[91,3] = PR[90,3] + 33.623;
   1:L PR[91] R[100]mm/sec CNT100;
   1:  PR[91,1] = PR[90,1] + 29.524;
   1:  PR[91,2] = PR[90,2] + 7.681;
   1:  PR[91,3] = PR[90,3] + 33.631;
   1:L PR[91] R[100]mm/sec CNT100;
   1:  PR[91,1] = PR[90,1] + 29.111;
   1:  PR[91,2] = PR[90,2] + 8.532;
   1:  PR[91,3] = PR[90,3] + 33.638;
   1:L PR[91] R[100]mm/sec CNT100;
   1:  PR[91,1] = PR[90,1] + 28.653;
   1:  PR[91,2] = PR[90,2] + 9.369;
   1:  PR[91,3] = PR[90,3] + 33.645;
   1:L PR[91] R[100]mm/sec CNT100;
   1:  PR[91,1] = PR[90,1] + 28.150;
   1:  PR[91,2] = PR[90,2] + 10.189;
   1:  PR[91,3] = PR[90,3] + 33.653;
   1:L PR[91] R[100]mm/sec CNT100;
   1:  PR[91,1] = PR[90,1] + 27.595;
   1:  PR[91,2] = PR[90,2] + 10.997;
   1:  PR[91,3] = PR[90,3] + 33.661;
   1:L PR[91] R[100]mm/sec CNT100;
   1:  PR[91,1] = PR[90,1] + 27.014;
   1:  PR[91,2] = PR[90,2] + 11.760;
   1:  PR[91,3] = PR[90,3] + 33.668;
   1:L PR[91] R[100]mm/sec CNT100;
   1:  PR[91,1] = PR[90,1] + 26.383;
   1:  PR[91,2] = PR[90,2] + 12.505;
   1:  PR[91,3] = PR[90,3] + 33.676;
   1:L PR[91] R[100]mm/sec CNT100;
   1:  PR[91,1] = PR[90,1] + 25.711;
   1:  PR[91,2] = PR[90,2] + 13.219;
   1:  PR[91,3] = PR[90,3] + 33.684;
   1:L PR[91] R[100]mm/sec CNT100;
   1:  PR[91,1] = PR[90,1] + 24.999;
   1:  PR[91,2] = PR[90,2] + 13.900;
   1:  PR[91,3] = PR[90,3] + 33.691;
   1:L PR[91] R[100]mm/sec CNT100;
   1:  PR[91,1] = PR[90,1] + 24.437;
   1:  PR[91,2] = PR[90,2] + 14.388;
   1:  PR[91,3] = PR[90,3] + 33.699;
   1:L PR[91] R[100]mm/sec CNT100;
   1:  PR[91,1] = PR[90,1] + 23.464;
   1:  PR[91,2] = PR[90,2] + 15.157;
   1:  PR[91,3] = PR[90,3] + 33.705;
   1:L PR[91] R[100]mm/sec CNT100;
   1:  PR[91,1] = PR[90,1] + 22.646;
   1:  PR[91,2] = PR[90,2] + 15.729;
   1:  PR[91,3] = PR[90,3] + 33.715;
   1:L PR[91] R[100]mm/sec CNT100;
   1:  PR[91,1] = PR[90,1] + 21.793;
   1:  PR[91,2] = PR[90,2] + 16.263;
   1:  PR[91,3] = PR[90,3] + 33.723;
   1:L PR[91] R[100]mm/sec CNT100;
   1:  PR[91,1] = PR[90,1] + 21.336;
   1:  PR[91,2] = PR[90,2] + 16.522;
   1:  PR[91,3] = PR[90,3] + 33.731;
   1:L PR[91] R[100]mm/sec CNT100;
   1:  PR[91,1] = PR[90,1] + 20.914;
   1:  PR[91,2] = PR[90,2] + 16.755;
   1:  PR[91,3] = PR[90,3] + 33.735;
   1:L PR[91] R[100]mm/sec CNT100;
   1:  PR[91,1] = PR[90,1] + 20.001;
   1:  PR[91,2] = PR[90,2] + 17.207;
   1:  PR[91,3] = PR[90,3] + 33.739;
   1:L PR[91] R[100]mm/sec CNT100;
   1:  PR[91,1] = PR[90,1] + 19.066;
   1:  PR[91,2] = PR[90,2] + 17.614;
   1:  PR[91,3] = PR[90,3] + 33.747;
   1:L PR[91] R[100]mm/sec CNT100;
   1:  PR[91,1] = PR[90,1] + 17.837;
   1:  PR[91,2] = PR[90,2] + 18.066;
   1:  PR[91,3] = PR[90,3] + 33.755;
   1:L PR[91] R[100]mm/sec CNT100;
   1:  PR[91,1] = PR[90,1] + 17.123;
   1:  PR[91,2] = PR[90,2] + 18.293;
   1:  PR[91,3] = PR[90,3] + 33.765;
   1:L PR[91] R[100]mm/sec CNT100;
   1:  PR[91,1] = PR[90,1] + 16.122;
   1:  PR[91,2] = PR[90,2] + 18.560;
   1:  PR[91,3] = PR[90,3] + 33.771;
   1:L PR[91] R[100]mm/sec CNT100;
   1:  PR[91,1] = PR[90,1] + 15.107;
   1:  PR[91,2] = PR[90,2] + 18.778;
   1:  PR[91,3] = PR[90,3] + 33.779;
   1:L PR[91] R[100]mm/sec CNT100;
   1:  PR[91,1] = PR[90,1] + 14.066;
   1:  PR[91,2] = PR[90,2] + 18.946;
   1:  PR[91,3] = PR[90,3] + 33.787;
   1:L PR[91] R[100]mm/sec CNT100;
   1:  PR[91,1] = PR[90,1] + 13.074;
   1:  PR[91,2] = PR[90,2] + 19.058;
   1:  PR[91,3] = PR[90,3] + 33.796;
   1:L PR[91] R[100]mm/sec CNT100;
   1:  PR[91,1] = PR[90,1] + 12.073;
   1:  PR[91,2] = PR[90,2] + 19.122;
   1:  PR[91,3] = PR[90,3] + 33.803;
   1:L PR[91] R[100]mm/sec CNT100;
   1:  PR[91,1] = PR[90,1] + 11.070;
   1:  PR[91,2] = PR[90,2] + 19.138;
   1:  PR[91,3] = PR[90,3] + 33.811;
   1:L PR[91] R[100]mm/sec CNT100;
   1:  PR[91,1] = PR[90,1] + 10.068;
   1:  PR[91,2] = PR[90,2] + 19.105;
   1:  PR[91,3] = PR[90,3] + 33.819;
   1:L PR[91] R[100]mm/sec CNT100;
   1:  PR[91,1] = PR[90,1] + 9.070;
   1:  PR[91,2] = PR[90,2] + 19.023;
   1:  PR[91,3] = PR[90,3] + 33.827;
   1:L PR[91] R[100]mm/sec CNT100;
   1:  PR[91,1] = PR[90,1] + 8.078;
   1:  PR[91,2] = PR[90,2] + 18.893;
   1:  PR[91,3] = PR[90,3] + 33.835;
   1:L PR[91] R[100]mm/sec CNT100;
   1:  PR[91,1] = PR[90,1] + 7.094;
   1:  PR[91,2] = PR[90,2] + 18.715;
   1:  PR[91,3] = PR[90,3] + 33.843;
   1:L PR[91] R[100]mm/sec CNT100;
   1:  PR[91,1] = PR[90,1] + 6.121;
   1:  PR[91,2] = PR[90,2] + 18.489;
   1:  PR[91,3] = PR[90,3] + 33.851;
   1:L PR[91] R[100]mm/sec CNT100;
   1:  PR[91,1] = PR[90,1] + 5.161;
   1:  PR[91,2] = PR[90,2] + 18.215;
   1:  PR[91,3] = PR[90,3] + 33.859;
   1:L PR[91] R[100]mm/sec CNT100;
   1:  PR[91,1] = PR[90,1] + 4.216;
   1:  PR[91,2] = PR[90,2] + 17.896;
   1:  PR[91,3] = PR[90,3] + 33.867;
   1:L PR[91] R[100]mm/sec CNT100;
   1:  PR[91,1] = PR[90,1] + 3.291;
   1:  PR[91,2] = PR[90,2] + 17.531;
   1:  PR[91,3] = PR[90,3] + 33.874;
   1:L PR[91] R[100]mm/sec CNT100;
   1:  PR[91,1] = PR[90,1] + 2.384;
   1:  PR[91,2] = PR[90,2] + 17.121;
   1:  PR[91,3] = PR[90,3] + 33.882;
   1:L PR[91] R[100]mm/sec CNT100;
   1:  PR[91,1] = PR[90,1] + 1.707;
   1:  PR[91,2] = PR[90,2] + 16.777;
   1:  PR[91,3] = PR[90,3] + 33.890;
   1:L PR[91] R[100]mm/sec CNT100;
   1:  PR[91,1] = PR[90,1] + 1.244;
   1:  PR[91,2] = PR[90,2] + 16.522;
   1:  PR[91,3] = PR[90,3] + 33.896;
   1:L PR[91] R[100]mm/sec CNT100;
   1:  PR[91,1] = PR[90,1] + 0.803;
   1:  PR[91,2] = PR[90,2] + 16.336;
   1:  PR[91,3] = PR[90,3] + 33.900;
   1:L PR[91] R[100]mm/sec CNT100;
   1:  PR[91,1] = PR[90,1] + 0.322;
   1:  PR[91,2] = PR[90,2] + 16.221;
   1:  PR[91,3] = PR[90,3] + 33.904;
   1:L PR[91] R[100]mm/sec CNT100;
   1:  PR[91,1] = PR[90,1] + -0.170;
   1:  PR[91,2] = PR[90,2] + 16.189;
   1:  PR[91,3] = PR[90,3] + 33.908;
   1:L PR[91] R[100]mm/sec CNT100;
   1:  PR[91,1] = PR[90,1] + -0.658;
   1:  PR[91,2] = PR[90,2] + 16.237;
   1:  PR[91,3] = PR[90,3] + 33.912;
   1:L PR[91] R[100]mm/sec CNT100;
   1:  PR[91,1] = PR[90,1] + -1.132;
   1:  PR[91,2] = PR[90,2] + 16.366;
   1:  PR[91,3] = PR[90,3] + 33.916;
   1:L PR[91] R[100]mm/sec CNT100;
   1:  PR[91,1] = PR[90,1] + -1.554;
   1:  PR[91,2] = PR[90,2] + 16.559;
   1:  PR[91,3] = PR[90,3] + 33.920;
   1:L PR[91] R[100]mm/sec CNT100;
   1:  PR[91,1] = PR[90,1] + -1.940;
   1:  PR[91,2] = PR[90,2] + 16.772;
   1:  PR[91,3] = PR[90,3] + 33.923;
   1:L PR[91] R[100]mm/sec CNT100;
   1:  PR[91,1] = PR[90,1] + -2.881;
   1:  PR[91,2] = PR[90,2] + 17.241;
   1:  PR[91,3] = PR[90,3] + 33.927;
   1:L PR[91] R[100]mm/sec CNT100;
   1:  PR[91,1] = PR[90,1] + -3.846;
   1:  PR[91,2] = PR[90,2] + 17.660;
   1:  PR[91,3] = PR[90,3] + 33.935;
   1:L PR[91] R[100]mm/sec CNT100;
   1:  PR[91,1] = PR[90,1] + -4.839;
   1:  PR[91,2] = PR[90,2] + 18.031;
   1:  PR[91,3] = PR[90,3] + 33.943;
   1:L PR[91] R[100]mm/sec CNT100;
   1:  PR[91,1] = PR[90,1] + -5.402;
   1:  PR[91,2] = PR[90,2] + 18.218;
   1:  PR[91,3] = PR[90,3] + 33.952;
   1:L PR[91] R[100]mm/sec CNT100;
   1:  PR[91,1] = PR[90,1] + -6.363;
   1:  PR[91,2] = PR[90,2] + 18.491;
   1:  PR[91,3] = PR[90,3] + 33.956;
   1:L PR[91] R[100]mm/sec CNT100;
   1:  PR[91,1] = PR[90,1] + -7.336;
   1:  PR[91,2] = PR[90,2] + 18.717;
   1:  PR[91,3] = PR[90,3] + 33.964;
   1:L PR[91] R[100]mm/sec CNT100;
   1:  PR[91,1] = PR[90,1] + -8.320;
   1:  PR[91,2] = PR[90,2] + 18.894;
   1:  PR[91,3] = PR[90,3] + 33.972;
   1:L PR[91] R[100]mm/sec CNT100;
   1:  PR[91,1] = PR[90,1] + -9.313;
   1:  PR[91,2] = PR[90,2] + 19.024;
   1:  PR[91,3] = PR[90,3] + 33.980;
   1:L PR[91] R[100]mm/sec CNT100;
   1:  PR[91,1] = PR[90,1] + -10.311;
   1:  PR[91,2] = PR[90,2] + 19.105;
   1:  PR[91,3] = PR[90,3] + 33.988;
   1:L PR[91] R[100]mm/sec CNT100;
   1:  PR[91,1] = PR[90,1] + -11.313;
   1:  PR[91,2] = PR[90,2] + 19.137;
   1:  PR[91,3] = PR[90,3] + 33.996;
   1:L PR[91] R[100]mm/sec CNT100;
   1:  PR[91,1] = PR[90,1] + -12.181;
   1:  PR[91,2] = PR[90,2] + 19.125;
   1:  PR[91,3] = PR[90,3] + 34.004;
   1:L PR[91] R[100]mm/sec CNT100;
   1:  PR[91,1] = PR[90,1] + -13.317;
   1:  PR[91,2] = PR[90,2] + 19.057;
   1:  PR[91,3] = PR[90,3] + 34.011;
   1:L PR[91] R[100]mm/sec CNT100;
   1:  PR[91,1] = PR[90,1] + -14.320;
   1:  PR[91,2] = PR[90,2] + 18.943;
   1:  PR[91,3] = PR[90,3] + 34.020;
   1:L PR[91] R[100]mm/sec CNT100;
   1:  PR[91,1] = PR[90,1] + -15.349;
   1:  PR[91,2] = PR[90,2] + 18.777;
   1:  PR[91,3] = PR[90,3] + 34.028;
   1:L PR[91] R[100]mm/sec CNT100;
   1:  PR[91,1] = PR[90,1] + -16.364;
   1:  PR[91,2] = PR[90,2] + 18.560;
   1:  PR[91,3] = PR[90,3] + 34.036;
   1:L PR[91] R[100]mm/sec CNT100;
   1:  PR[91,1] = PR[90,1] + -17.364;
   1:  PR[91,2] = PR[90,2] + 18.293;
   1:  PR[91,3] = PR[90,3] + 34.044;
   1:L PR[91] R[100]mm/sec CNT100;
   1:  PR[91,1] = PR[90,1] + -18.345;
   1:  PR[91,2] = PR[90,2] + 17.978;
   1:  PR[91,3] = PR[90,3] + 34.052;
   1:L PR[91] R[100]mm/sec CNT100;
   1:  PR[91,1] = PR[90,1] + -19.304;
   1:  PR[91,2] = PR[90,2] + 17.615;
   1:  PR[91,3] = PR[90,3] + 34.060;
   1:L PR[91] R[100]mm/sec CNT100;
   1:  PR[91,1] = PR[90,1] + -20.241;
   1:  PR[91,2] = PR[90,2] + 17.207;
   1:  PR[91,3] = PR[90,3] + 34.068;
   1:L PR[91] R[100]mm/sec CNT100;
   1:  PR[91,1] = PR[90,1] + -21.152;
   1:  PR[91,2] = PR[90,2] + 16.754;
   1:  PR[91,3] = PR[90,3] + 34.076;
   1:L PR[91] R[100]mm/sec CNT100;
   1:  PR[91,1] = PR[90,1] + -22.034;
   1:  PR[91,2] = PR[90,2] + 16.260;
   1:  PR[91,3] = PR[90,3] + 34.084;
   1:L PR[91] R[100]mm/sec CNT100;
   1:  PR[91,1] = PR[90,1] + -22.888;
   1:  PR[91,2] = PR[90,2] + 15.724;
   1:  PR[91,3] = PR[90,3] + 34.092;
   1:L PR[91] R[100]mm/sec CNT100;
   1:  PR[91,1] = PR[90,1] + -23.178;
   1:  PR[91,2] = PR[90,2] + 15.523;
   1:  PR[91,3] = PR[90,3] + 34.100;
   1:L PR[91] R[100]mm/sec CNT100;
   1:  PR[91,1] = PR[90,1] + -23.705;
   1:  PR[91,2] = PR[90,2] + 15.152;
   1:  PR[91,3] = PR[90,3] + 34.103;
   1:L PR[91] R[100]mm/sec CNT100;
   1:  PR[91,1] = PR[90,1] + -24.491;
   1:  PR[91,2] = PR[90,2] + 14.542;
   1:  PR[91,3] = PR[90,3] + 34.108;
   1:L PR[91] R[100]mm/sec CNT100;
   1:  PR[91,1] = PR[90,1] + -25.240;
   1:  PR[91,2] = PR[90,2] + 13.896;
   1:  PR[91,3] = PR[90,3] + 34.116;
   1:L PR[91] R[100]mm/sec CNT100;
   1:  PR[91,1] = PR[90,1] + -25.951;
   1:  PR[91,2] = PR[90,2] + 13.218;
   1:  PR[91,3] = PR[90,3] + 34.124;
   1:L PR[91] R[100]mm/sec CNT100;
   1:  PR[91,1] = PR[90,1] + -26.623;
   1:  PR[91,2] = PR[90,2] + 12.507;
   1:  PR[91,3] = PR[90,3] + 34.132;
   1:L PR[91] R[100]mm/sec CNT100;
   1:  PR[91,1] = PR[90,1] + -27.253;
   1:  PR[91,2] = PR[90,2] + 11.765;
   1:  PR[91,3] = PR[90,3] + 34.139;
   1:L PR[91] R[100]mm/sec CNT100;
   1:  PR[91,1] = PR[90,1] + -27.849;
   1:  PR[91,2] = PR[90,2] + 10.985;
   1:  PR[91,3] = PR[90,3] + 34.147;
   1:L PR[91] R[100]mm/sec CNT100;
   1:  PR[91,1] = PR[90,1] + -28.381;
   1:  PR[91,2] = PR[90,2] + 10.209;
   1:  PR[91,3] = PR[90,3] + 34.155;
   1:L PR[91] R[100]mm/sec CNT100;
   1:  PR[91,1] = PR[90,1] + -28.881;
   1:  PR[91,2] = PR[90,2] + 9.395;
   1:  PR[91,3] = PR[90,3] + 34.162;
   1:L PR[91] R[100]mm/sec CNT100;
   1:  PR[91,1] = PR[90,1] + -29.338;
   1:  PR[91,2] = PR[90,2] + 8.558;
   1:  PR[91,3] = PR[90,3] + 34.170;
   1:L PR[91] R[100]mm/sec CNT100;
   1:  PR[91,1] = PR[90,1] + -29.750;
   1:  PR[91,2] = PR[90,2] + 7.705;
   1:  PR[91,3] = PR[90,3] + 34.177;
   1:L PR[91] R[100]mm/sec CNT100;
